KUKA KRL program: PPR_fullpath_2mm_split3.src

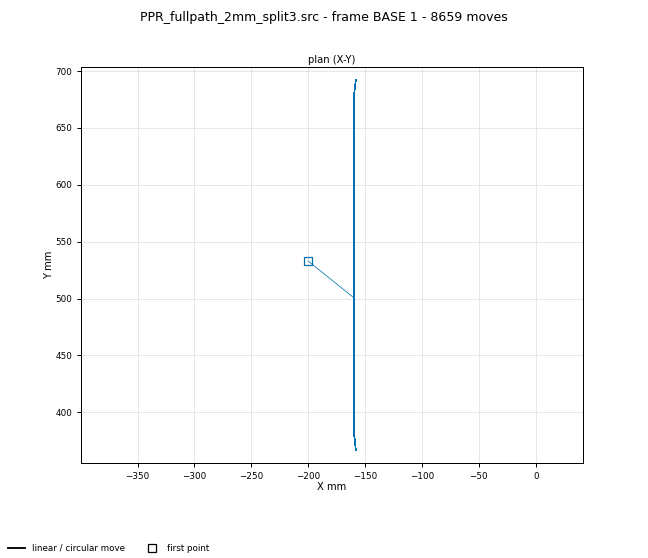
[picture p0: tool path of PPR_fullpath_2mm_split3.src in frame BASE 1, 8659 of 8660 moves have a stored position in this frame; points joined in program order, loops and branches not executed]
&ACCESS RVEO
&REL 11
&PARAM TEMPLATE = C:\KRC\Roboter\Template\vorgabe
&PARAM EDITMASK = *
DEF variable_helical2( )
;FOLD INI
  ;FOLD BASISTECH INI
    GLOBAL INTERRUPT DECL 3 WHEN $STOPMESS==TRUE DO IR_STOPM ( )
    INTERRUPT ON 3
    BAS (#INITMOV,0 )
  ;ENDFOLD (BASISTECH INI)
 ;FOLD USER INI


    ;Make your modifications here
  ;ENDFOLD (USER INI)
;ENDFOLD (INI)
ACTION(#AXIS_RESET,34,1000,#NOERROR,ERROR_CODE)
;FOLD PTP HOME  Vel= 100 % DEFAULT;%{PE}%MKUKATPBASIS,%CMOVE,%VPTP,%P 1:PTP, 2:HOME, 3:, 5:100, 7:DEFAULT
$BWDSTART = FALSE
PDAT_ACT=PDEFAULT
FDAT_ACT=FHOME
BAS (#PTP_PARAMS,100 )
$H_POS=XHOME
PTP  XHOME
;ENDFOLD
BAS(#TOOL,1)
BAS(#BASE,1)
$VEL_AXIS[1]=100
$VEL_AXIS[2]=100
$VEL_AXIS[3]=100
$VEL_AXIS[4]=100
$VEL_AXIS[5]=100
$VEL_AXIS[6]=100
$VEL_EXTAX[1]=100
$VEL_EXTAX[2]=100

$ACC_AXIS[1]=100
$ACC_AXIS[2]=100
$ACC_AXIS[3]=100
$ACC_AXIS[4]=100
$ACC_AXIS[5]=100
$ACC_AXIS[6]=100
$ACC_EXTAX[1]=100
$ACC_EXTAX[2]=100

SLIN {X  -200.000, Y  +533.000, Z    +0.000, A    +0.000, E1    +0.000, E3    +0.000, E4    +0.000}

SLIN {X  -160.000, Y  +500.804, Z    +0.000, E1   +21.423, E3  -369.741}
HALT
SPLINE
SPL {X  -160.000, Y  +497.229, Z    +0.000, E1   +21.403, E3  -350.308}
SPL {X  -160.000, Y  +493.901, Z    +0.000, E1   +21.409, E3  -332.289}
SPL {X  -160.000, Y  +490.791, Z    +0.000, E1   +21.400, E3  -315.416}
SPL {X  -160.000, Y  +487.647, Z    +0.000, E1   +21.401, E3  -298.370}
SPL {X  -160.000, Y  +484.273, Z    +0.000, E1   +21.408, E3  -280.090}
SPL {X  -160.000, Y  +481.093, Z    +0.000, E1   +21.389, E3  -262.781}
SPL {X  -160.000, Y  +478.021, Z    +0.000, E1   +21.401, E3  -246.174}
SPL {X  -160.000, Y  +474.639, Z    +0.000, E1   +21.410, E3  -227.883}
SPL {X  -160.000, Y  +471.343, Z    +0.000, E1   +21.399, E3  -209.981}
SPL {X  -160.000, Y  +468.133, Z    +0.000, E1   +21.402, E3  -192.589}
SPL {X  -160.000, Y  +464.638, Z    +0.000, E1   +21.421, E3  -173.740}
SPL {X  -160.000, Y  +461.045, Z    +0.000, E1   +21.424, E3  -154.326}
SPL {X  -160.000, Y  +457.606, Z    +0.000, E1   +21.413, E3  -135.616}
SPL {X  -160.000, Y  +454.417, Z    +0.000, E1   +21.401, E3  -118.308}
SPL {X  -160.000, Y  +451.425, Z    +0.000, E1   +21.404, E3  -102.086}
SPL {X  -160.000, Y  +448.039, Z    +0.000, E1   +21.417, E3   -83.793}
SPL {X  -160.000, Y  +444.787, Z    +0.000, E1   +21.414, E3   -66.238}
SPL {X  -160.000, Y  +441.637, Z    +0.000, E1   +21.431, E3   -49.260}
SPL {X  -160.000, Y  +438.199, Z    +0.000, E1   +21.432, E3   -30.656}
SPL {X  -160.000, Y  +434.875, Z    +0.000, E1   +21.424, E3   -12.616}
SPL {X  -160.000, Y  +431.689, Z    +0.000, E1   +21.423, E3    +4.632}
SPL {X  -160.000, Y  +428.451, Z    +0.000, E1   +21.430, E3   +22.112}
SPL {X  -160.000, Y  +425.120, Z    +0.000, E1   +21.430, E3   +40.176}
SPL {X  -160.000, Y  +421.671, Z    +0.000, E1   +21.430, E3   +58.860}
SPL {X  -160.000, Y  +418.225, Z    +0.000, E1   +21.425, E3   +77.542}
SPL {X  -160.000, Y  +414.956, Z    +0.000, E1   +21.424, E3   +95.222}
SPL {X  -160.000, Y  +411.834, Z    +0.000, E1   +21.420, E3  +112.140}
SPL {X  -160.000, Y  +408.570, Z    +0.000, E1   +21.432, E3  +129.749}
SPL {X  -160.000, Y  +405.237, Z    +0.000, E1   +21.432, E3  +147.778}
SPL {X  -160.000, Y  +402.004, Z    +0.000, E1   +21.424, E3  +165.353}
SPL {X  -160.000, Y  +398.626, Z    +0.000, E1   +21.425, E3  +183.659}
SPL {X  -160.000, Y  +395.405, Z    +0.000, E1   +21.422, E3  +201.077}
SPL {X  -160.000, Y  +392.641, Z    +0.000, E1   +21.407, E3  +216.075}
SPL {X  -159.989, Y  +390.129, Z    +0.000, E1   +21.406, E3  +229.716}
SPL {X  -159.932, Y  +387.337, Z    +0.000, E1   +21.403, E3  +244.912}
SPL {X  -159.823, Y  +384.478, Z    +0.000, E1   +21.379, E3  +260.575}
SPL {X  -159.660, Y  +381.581, Z    +0.000, E1   +21.363, E3  +276.463}
SPL {X  -159.452, Y  +378.773, Z    +0.000, E1   +21.330, E3  +291.910}
SPL {X  -159.222, Y  +376.244, Z    +0.000, E1   +21.297, E3  +305.872}
SPL {X  -158.814, Y  +372.556, Z    +0.000, E1   +21.316, E3  +326.139}
SPL {X  -158.301, Y  +368.743, Z    +0.000, E1   +21.199, E3  +347.461}
SPL {X  -157.981, Y  +366.660, Z    +0.000, E1   +19.986, E3  +370.429}
ENDSPLINE

SPLINE
SPL {X  -158.491, Y  +370.077, Z    +0.000, E1   +15.910, E3  +395.442}
SPL {X  -159.771, Y  +383.450, Z    +0.000, E1    +6.314, E3  +418.597}
SPL {X  -160.000, Y  +392.463, Z    +0.000, E1    +0.112, E3  +425.104}
SPL {X  -160.000, Y  +399.874, Z    +0.000, E1    -5.508, E3  +429.606}
SPL {X  -160.000, Y  +411.622, Z    +0.000, E1   -13.815, E3  +441.726}
SPL {X  -160.000, Y  +419.836, Z    +0.000, E1   -18.198, E3  +456.900}
SPL {X  -160.000, Y  +430.523, Z    +0.000, E1   -21.710, E3  +487.100}
SPL {X  -160.000, Y  +433.426, Z    +0.000, E1   -21.735, E3  +502.515}
SPL {X  -160.000, Y  +436.131, Z    +0.000, E1   -21.710, E3  +516.989}
SPL {X  -160.000, Y  +439.046, Z    +0.000, E1   -21.732, E3  +532.483}
SPL {X  -160.000, Y  +442.009, Z    +0.000, E1   -21.719, E3  +548.305}
SPL {X  -160.000, Y  +444.891, Z    +0.000, E1   -21.724, E3  +563.661}
SPL {X  -160.000, Y  +449.017, Z    +0.000, E1   -21.792, E3  +585.452}
SPL {X  -160.000, Y  +452.864, Z    +0.000, E1   -21.730, E3  +606.070}
SPL {X  -160.000, Y  +455.470, Z    +0.000, E1   -21.722, E3  +619.959}
SPL {X  -160.000, Y  +458.295, Z    +0.000, E1   -21.738, E3  +634.980}
SPL {X  -160.000, Y  +461.133, Z    +0.000, E1   -21.720, E3  +650.162}
SPL {X  -160.000, Y  +464.458, Z    +0.000, E1   -21.770, E3  +667.681}
SPL {X  -160.000, Y  +468.250, Z    +0.000, E1   -21.764, E3  +687.834}
SPL {X  -160.000, Y  +472.226, Z    +0.000, E1   -21.782, E3  +708.993}
SPL {X  -160.000, Y  +476.333, Z    +0.000, E1   -21.767, E3  +730.907}
SPL {X  -160.000, Y  +480.244, Z    +0.000, E1   -21.765, E3  +751.772}
SPL {X  -160.000, Y  +484.301, Z    +0.000, E1   -21.775, E3  +773.300}
SPL {X  -160.000, Y  +488.201, Z    +0.000, E1   -21.768, E3  +794.060}
SPL {X  -160.000, Y  +492.394, Z    +0.000, E1   -21.802, E3  +816.234}
SPL {X  -160.000, Y  +496.781, Z    +0.000, E1   -21.798, E3  +839.546}
SPL {X  -160.000, Y  +501.083, Z    +0.000, E1   -21.796, E3  +862.476}
SPL {X  -160.000, Y  +504.917, Z    +0.000, E1   -21.764, E3  +882.980}
SPL {X  -160.000, Y  +508.886, Z    +0.000, E1   -21.791, E3  +904.066}
SPL {X  -160.000, Y  +513.057, Z    +0.000, E1   -21.767, E3  +926.374}
SPL {X  -160.000, Y  +517.221, Z    +0.000, E1   -21.778, E3  +948.527}
SPL {X  -160.000, Y  +521.677, Z    +0.000, E1   -21.781, E3  +972.288}
SPL {X  -160.000, Y  +525.729, Z    +0.000, E1   -21.753, E3  +993.927}
SPL {X  -160.000, Y  +529.456, Z    +0.000, E1   -21.766, E3 +1013.706}
SPL {X  -160.000, Y  +533.608, Z    +0.000, E1   -21.776, E3 +1035.837}
SPL {X  -160.000, Y  +538.227, Z    +0.000, E1   -21.794, E3 +1060.369}
SPL {X  -160.000, Y  +542.483, Z    +0.000, E1   -21.764, E3 +1083.095}
SPL {X  -160.000, Y  +546.194, Z    +0.000, E1   -21.754, E3 +1102.911}
SPL {X  -160.000, Y  +550.131, Z    +0.000, E1   -21.771, E3 +1123.847}
SPL {X  -160.000, Y  +554.462, Z    +0.000, E1   -21.777, E3 +1146.901}
SPL {X  -160.000, Y  +558.542, Z    +0.000, E1   -21.758, E3 +1168.673}
SPL {X  -160.000, Y  +562.615, Z    +0.000, E1   -21.776, E3 +1190.329}
SPL {X  -160.000, Y  +566.764, Z    +0.000, E1   -21.764, E3 +1212.454}
SPL {X  -160.000, Y  +570.657, Z    +0.000, E1   -21.758, E3 +1233.201}
SPL {X  -160.000, Y  +574.688, Z    +0.000, E1   -21.771, E3 +1254.644}
SPL {X  -160.000, Y  +578.864, Z    +0.000, E1   -21.770, E3 +1276.895}
SPL {X  -160.000, Y  +582.807, Z    +0.000, E1   -21.754, E3 +1297.949}
SPL {X  -160.000, Y  +586.993, Z    +0.000, E1   -21.779, E3 +1320.185}
SPL {X  -160.000, Y  +591.368, Z    +0.000, E1   -21.775, E3 +1343.472}
SPL {X  -160.000, Y  +595.703, Z    +0.000, E1   -21.775, E3 +1366.581}
SPL {X  -160.000, Y  +599.558, Z    +0.000, E1   -21.748, E3 +1387.159}
SPL {X  -160.000, Y  +603.126, Z    +0.000, E1   -21.757, E3 +1406.138}
SPL {X  -160.000, Y  +607.107, Z    +0.000, E1   -21.766, E3 +1427.364}
SPL {X  -160.000, Y  +611.246, Z    +0.000, E1   -21.760, E3 +1449.437}
SPL {X  -160.000, Y  +615.151, Z    +0.000, E1   -21.752, E3 +1470.250}
SPL {X  -160.000, Y  +618.728, Z    +0.000, E1   -21.747, E3 +1489.312}
SPL {X  -160.000, Y  +622.318, Z    +0.000, E1   -21.753, E3 +1508.427}
SPL {X  -160.000, Y  +625.877, Z    +0.000, E1   -21.745, E3 +1527.405}
SPL {X  -160.000, Y  +629.892, Z    +0.000, E1   -21.777, E3 +1548.729}
SPL {X  -160.000, Y  +634.024, Z    +0.000, E1   -21.756, E3 +1570.779}
SPL {X  -160.000, Y  +637.661, Z    +0.000, E1   -21.748, E3 +1590.170}
SPL {X  -160.000, Y  +641.244, Z    +0.000, E1   -21.752, E3 +1609.241}
SPL {X  -160.000, Y  +645.120, Z    +0.000, E1   -21.762, E3 +1629.873}
SPL {X  -160.000, Y  +649.214, Z    +0.000, E1   -21.766, E3 +1651.661}
SPL {X  -160.000, Y  +653.188, Z    +0.000, E1   -21.771, E3 +1672.724}
SPL {X  -160.000, Y  +656.905, Z    +0.000, E1   -21.769, E3 +1692.499}
SPL {X  -160.000, Y  +660.685, Z    +0.000, E1   -21.769, E3 +1712.667}
SPL {X  -160.000, Y  +664.985, Z    +0.000, E1   -21.790, E3 +1735.520}
SPL {X  -159.993, Y  +669.170, Z    +0.000, E1   -21.763, E3 +1757.878}
SPL {X  -159.916, Y  +672.869, Z    +0.000, E1   -21.755, E3 +1777.623}
SPL {X  -159.752, Y  +676.610, Z    +0.000, E1   -21.740, E3 +1797.698}
SPL {X  -159.478, Y  +680.618, Z    +0.000, E1   -21.719, E3 +1819.297}
SPL {X  -159.108, Y  +684.576, Z    +0.000, E1   -21.664, E3 +1840.767}
SPL {X  -158.638, Y  +688.530, Z    +0.000, E1   -21.617, E3 +1862.288}
SPL {X  -158.097, Y  +692.303, Z    +0.000, E1   -21.529, E3 +1883.006}
ENDSPLINE

SPLINE
SPL {X  -158.264, Y  +691.203, Z    +0.000, E1   -17.264, E3 +1919.751}
SPL {X  -159.000, Y  +685.560, Z    +0.000, E1   -12.398, E3 +1940.927}
SPL {X  -159.924, Y  +672.625, Z    +0.000, E1    -3.689, E3 +1955.944}
SPL {X  -160.000, Y  +663.203, Z    +0.000, E1    +3.155, E3 +1962.598}
SPL {X  -160.000, Y  +652.103, Z    +0.000, E1   +11.247, E3 +1974.268}
SPL {X  -160.000, Y  +641.822, Z    +0.000, E1   +17.059, E3 +1993.642}
SPL {X  -160.000, Y  +631.293, Z    +0.000, E1   +20.354, E3 +2027.522}
SPL {X  -160.000, Y  +627.542, Z    +0.000, E1   +20.380, E3 +2048.929}
SPL {X  -160.000, Y  +623.532, Z    +0.000, E1   +20.378, E3 +2071.894}
SPL {X  -160.000, Y  +619.329, Z    +0.000, E1   +20.391, E3 +2095.932}
SPL {X  -160.000, Y  +614.967, Z    +0.000, E1   +20.392, E3 +2120.912}
SPL {X  -160.000, Y  +611.206, Z    +0.000, E1   +20.351, E3 +2142.583}
SPL {X  -160.000, Y  +607.824, Z    +0.000, E1   +20.354, E3 +2162.004}
SPL {X  -160.000, Y  +603.899, Z    +0.000, E1   +20.373, E3 +2184.454}
SPL {X  -160.000, Y  +599.617, Z    +0.000, E1   +20.384, E3 +2208.948}
SPL {X  -160.000, Y  +595.532, Z    +0.000, E1   +20.373, E3 +2232.308}
SPL {X  -160.000, Y  +591.705, Z    +0.000, E1   +20.373, E3 +2254.233}
SPL {X  -160.000, Y  +588.037, Z    +0.000, E1   +20.359, E3 +2275.320}
SPL {X  -160.000, Y  +584.320, Z    +0.000, E1   +20.364, E3 +2296.622}
SPL {X  -160.000, Y  +580.616, Z    +0.000, E1   +20.357, E3 +2317.849}
SPL {X  -160.000, Y  +577.083, Z    +0.000, E1   +20.358, E3 +2338.097}
SPL {X  -160.000, Y  +573.158, Z    +0.000, E1   +20.377, E3 +2360.549}
SPL {X  -160.000, Y  +568.802, Z    +0.000, E1   +20.385, E3 +2385.501}
SPL {X  -160.000, Y  +564.937, Z    +0.000, E1   +20.350, E3 +2407.722}
SPL {X  -160.000, Y  +561.213, Z    +0.000, E1   +20.372, E3 +2429.008}
SPL {X  -160.000, Y  +557.320, Z    +0.000, E1   +20.363, E3 +2451.335}
SPL {X  -160.000, Y  +553.712, Z    +0.000, E1   +20.355, E3 +2472.034}
SPL {X  -160.000, Y  +550.040, Z    +0.000, E1   +20.360, E3 +2493.072}
SPL {X  -160.000, Y  +546.180, Z    +0.000, E1   +20.370, E3 +2515.128}
SPL {X  -160.000, Y  +542.032, Z    +0.000, E1   +20.384, E3 +2538.867}
SPL {X  -160.000, Y  +537.870, Z    +0.000, E1   +20.372, E3 +2562.743}
SPL {X  -160.000, Y  +534.086, Z    +0.000, E1   +20.356, E3 +2584.497}
SPL {X  -160.000, Y  +530.164, Z    +0.000, E1   +20.382, E3 +2606.846}
SPL {X  -160.000, Y  +527.505, Z    +0.000, E1   +20.318, E3 +2622.220}
SPL {X  -160.000, Y  +511.620, Z    +0.000, E1   +28.365, E3 +2632.683}
SPL {X  -160.000, Y  +507.906, Z    +0.000, E1   +28.152, E3 +2649.078}
SPL {X  -160.000, Y  +506.085, Z    +0.000, E1   +26.146, E3 +2671.538}
SPL {X  -160.000, Y  +504.342, Z    +0.000, E1   +24.109, E3 +2695.053}
SPL {X  -160.000, Y  +503.002, Z    +0.000, E1   +22.325, E3 +2716.058}
SPL {X  -160.000, Y  +500.783, Z    +0.000, E1   +21.421, E3 +2735.647}
SPL {X  -160.000, Y  +497.229, Z    +0.000, E1   +21.403, E3 +2754.956}
SPL {X  -160.000, Y  +493.901, Z    +0.000, E1   +21.409, E3 +2772.975}
SPL {X  -160.000, Y  +490.791, Z    +0.000, E1   +21.400, E3 +2789.848}
SPL {X  -160.000, Y  +487.647, Z    +0.000, E1   +21.401, E3 +2806.894}
SPL {X  -160.000, Y  +484.273, Z    +0.000, E1   +21.408, E3 +2825.174}
SPL {X  -160.000, Y  +481.093, Z    +0.000, E1   +21.389, E3 +2842.483}
SPL {X  -160.000, Y  +478.021, Z    +0.000, E1   +21.401, E3 +2859.089}
SPL {X  -160.000, Y  +474.639, Z    +0.000, E1   +21.410, E3 +2877.381}
SPL {X  -160.000, Y  +471.343, Z    +0.000, E1   +21.399, E3 +2895.283}
SPL {X  -160.000, Y  +468.133, Z    +0.000, E1   +21.402, E3 +2912.674}
SPL {X  -160.000, Y  +464.638, Z    +0.000, E1   +21.421, E3 +2931.523}
SPL {X  -160.000, Y  +461.045, Z    +0.000, E1   +21.424, E3 +2950.937}
SPL {X  -160.000, Y  +457.606, Z    +0.000, E1   +21.413, E3 +2969.647}
SPL {X  -160.000, Y  +454.417, Z    +0.000, E1   +21.401, E3 +2986.956}
SPL {X  -160.000, Y  +451.425, Z    +0.000, E1   +21.404, E3 +3003.177}
SPL {X  -160.000, Y  +448.039, Z    +0.000, E1   +21.417, E3 +3021.470}
SPL {X  -160.000, Y  +444.787, Z    +0.000, E1   +21.414, E3 +3039.025}
SPL {X  -160.000, Y  +441.637, Z    +0.000, E1   +21.431, E3 +3056.004}
SPL {X  -160.000, Y  +438.199, Z    +0.000, E1   +21.432, E3 +3074.607}
SPL {X  -160.000, Y  +434.875, Z    +0.000, E1   +21.424, E3 +3092.647}
SPL {X  -160.000, Y  +431.689, Z    +0.000, E1   +21.423, E3 +3109.896}
SPL {X  -160.000, Y  +428.451, Z    +0.000, E1   +21.430, E3 +3127.375}
SPL {X  -160.000, Y  +425.120, Z    +0.000, E1   +21.430, E3 +3145.440}
SPL {X  -160.000, Y  +421.671, Z    +0.000, E1   +21.430, E3 +3164.123}
SPL {X  -160.000, Y  +418.225, Z    +0.000, E1   +21.425, E3 +3182.805}
SPL {X  -160.000, Y  +414.956, Z    +0.000, E1   +21.424, E3 +3200.486}
SPL {X  -160.000, Y  +411.834, Z    +0.000, E1   +21.420, E3 +3217.404}
SPL {X  -160.000, Y  +408.570, Z    +0.000, E1   +21.432, E3 +3235.013}
SPL {X  -160.000, Y  +405.237, Z    +0.000, E1   +21.432, E3 +3253.041}
SPL {X  -160.000, Y  +402.004, Z    +0.000, E1   +21.424, E3 +3270.617}
SPL {X  -160.000, Y  +398.626, Z    +0.000, E1   +21.425, E3 +3288.923}
SPL {X  -160.000, Y  +395.405, Z    +0.000, E1   +21.422, E3 +3306.340}
SPL {X  -160.000, Y  +392.641, Z    +0.000, E1   +21.407, E3 +3321.339}
SPL {X  -159.989, Y  +390.129, Z    +0.000, E1   +21.406, E3 +3334.980}
SPL {X  -159.932, Y  +387.337, Z    +0.000, E1   +21.403, E3 +3350.175}
SPL {X  -159.823, Y  +384.478, Z    +0.000, E1   +21.379, E3 +3365.838}
SPL {X  -159.660, Y  +381.581, Z    +0.000, E1   +21.363, E3 +3381.727}
SPL {X  -159.452, Y  +378.773, Z    +0.000, E1   +21.330, E3 +3397.173}
SPL {X  -159.222, Y  +376.244, Z    +0.000, E1   +21.297, E3 +3411.136}
SPL {X  -158.814, Y  +372.556, Z    +0.000, E1   +21.316, E3 +3431.403}
SPL {X  -158.301, Y  +368.743, Z    +0.000, E1   +21.199, E3 +3452.725}
SPL {X  -157.981, Y  +366.660, Z    +0.000, E1   +19.986, E3 +3475.692}
ENDSPLINE

SPLINE
SPL {X  -158.491, Y  +370.077, Z    +0.000, E1   +15.910, E3 +3500.705}
SPL {X  -159.771, Y  +383.450, Z    +0.000, E1    +6.314, E3 +3523.861}
SPL {X  -160.000, Y  +392.463, Z    +0.000, E1    +0.112, E3 +3530.367}
SPL {X  -160.000, Y  +399.874, Z    +0.000, E1    -5.508, E3 +3534.870}
SPL {X  -160.000, Y  +411.622, Z    +0.000, E1   -13.815, E3 +3546.990}
SPL {X  -160.000, Y  +419.836, Z    +0.000, E1   -18.198, E3 +3562.163}
SPL {X  -160.000, Y  +430.523, Z    +0.000, E1   -21.710, E3 +3592.364}
SPL {X  -160.000, Y  +433.426, Z    +0.000, E1   -21.735, E3 +3607.778}
SPL {X  -160.000, Y  +436.131, Z    +0.000, E1   -21.710, E3 +3622.253}
SPL {X  -160.000, Y  +439.046, Z    +0.000, E1   -21.732, E3 +3637.746}
SPL {X  -160.000, Y  +442.009, Z    +0.000, E1   -21.719, E3 +3653.568}
SPL {X  -160.000, Y  +444.891, Z    +0.000, E1   -21.724, E3 +3668.924}
SPL {X  -160.000, Y  +449.017, Z    +0.000, E1   -21.792, E3 +3690.716}
SPL {X  -160.000, Y  +452.864, Z    +0.000, E1   -21.730, E3 +3711.333}
SPL {X  -160.000, Y  +455.470, Z    +0.000, E1   -21.722, E3 +3725.222}
SPL {X  -160.000, Y  +458.295, Z    +0.000, E1   -21.738, E3 +3740.243}
SPL {X  -160.000, Y  +461.133, Z    +0.000, E1   -21.720, E3 +3755.426}
SPL {X  -160.000, Y  +464.458, Z    +0.000, E1   -21.770, E3 +3772.945}
SPL {X  -160.000, Y  +468.250, Z    +0.000, E1   -21.764, E3 +3793.098}
SPL {X  -160.000, Y  +472.226, Z    +0.000, E1   -21.782, E3 +3814.256}
SPL {X  -160.000, Y  +476.333, Z    +0.000, E1   -21.767, E3 +3836.171}
SPL {X  -160.000, Y  +480.244, Z    +0.000, E1   -21.765, E3 +3857.035}
SPL {X  -160.000, Y  +484.301, Z    +0.000, E1   -21.775, E3 +3878.564}
SPL {X  -160.000, Y  +488.201, Z    +0.000, E1   -21.768, E3 +3899.324}
SPL {X  -160.000, Y  +492.394, Z    +0.000, E1   -21.802, E3 +3921.498}
SPL {X  -160.000, Y  +496.781, Z    +0.000, E1   -21.798, E3 +3944.809}
SPL {X  -160.000, Y  +501.083, Z    +0.000, E1   -21.796, E3 +3967.739}
SPL {X  -160.000, Y  +504.917, Z    +0.000, E1   -21.764, E3 +3988.244}
SPL {X  -160.000, Y  +508.886, Z    +0.000, E1   -21.791, E3 +4009.330}
SPL {X  -160.000, Y  +513.057, Z    +0.000, E1   -21.767, E3 +4031.637}
SPL {X  -160.000, Y  +517.221, Z    +0.000, E1   -21.778, E3 +4053.790}
SPL {X  -160.000, Y  +521.677, Z    +0.000, E1   -21.781, E3 +4077.551}
SPL {X  -160.000, Y  +525.729, Z    +0.000, E1   -21.753, E3 +4099.191}
SPL {X  -160.000, Y  +529.456, Z    +0.000, E1   -21.766, E3 +4118.970}
SPL {X  -160.000, Y  +533.608, Z    +0.000, E1   -21.776, E3 +4141.100}
SPL {X  -160.000, Y  +538.227, Z    +0.000, E1   -21.794, E3 +4165.633}
SPL {X  -160.000, Y  +542.483, Z    +0.000, E1   -21.764, E3 +4188.358}
SPL {X  -160.000, Y  +546.194, Z    +0.000, E1   -21.754, E3 +4208.174}
SPL {X  -160.000, Y  +550.131, Z    +0.000, E1   -21.771, E3 +4229.110}
SPL {X  -160.000, Y  +554.462, Z    +0.000, E1   -21.777, E3 +4252.164}
SPL {X  -160.000, Y  +558.542, Z    +0.000, E1   -21.758, E3 +4273.937}
SPL {X  -160.000, Y  +562.615, Z    +0.000, E1   -21.776, E3 +4295.593}
SPL {X  -160.000, Y  +566.764, Z    +0.000, E1   -21.764, E3 +4317.718}
SPL {X  -160.000, Y  +570.657, Z    +0.000, E1   -21.758, E3 +4338.465}
SPL {X  -160.000, Y  +574.688, Z    +0.000, E1   -21.771, E3 +4359.908}
SPL {X  -160.000, Y  +578.864, Z    +0.000, E1   -21.770, E3 +4382.159}
SPL {X  -160.000, Y  +582.807, Z    +0.000, E1   -21.754, E3 +4403.213}
SPL {X  -160.000, Y  +586.993, Z    +0.000, E1   -21.779, E3 +4425.448}
SPL {X  -160.000, Y  +591.368, Z    +0.000, E1   -21.775, E3 +4448.735}
SPL {X  -160.000, Y  +595.703, Z    +0.000, E1   -21.775, E3 +4471.845}
SPL {X  -160.000, Y  +599.558, Z    +0.000, E1   -21.748, E3 +4492.422}
SPL {X  -160.000, Y  +603.126, Z    +0.000, E1   -21.757, E3 +4511.402}
SPL {X  -160.000, Y  +607.107, Z    +0.000, E1   -21.766, E3 +4532.627}
SPL {X  -160.000, Y  +611.246, Z    +0.000, E1   -21.760, E3 +4554.700}
SPL {X  -160.000, Y  +615.151, Z    +0.000, E1   -21.752, E3 +4575.514}
SPL {X  -160.000, Y  +618.728, Z    +0.000, E1   -21.747, E3 +4594.576}
SPL {X  -160.000, Y  +622.318, Z    +0.000, E1   -21.753, E3 +4613.690}
SPL {X  -160.000, Y  +625.877, Z    +0.000, E1   -21.745, E3 +4632.669}
SPL {X  -160.000, Y  +629.892, Z    +0.000, E1   -21.777, E3 +4653.992}
SPL {X  -160.000, Y  +634.024, Z    +0.000, E1   -21.756, E3 +4676.043}
SPL {X  -160.000, Y  +637.661, Z    +0.000, E1   -21.748, E3 +4695.433}
SPL {X  -160.000, Y  +641.244, Z    +0.000, E1   -21.752, E3 +4714.504}
SPL {X  -160.000, Y  +645.120, Z    +0.000, E1   -21.762, E3 +4735.137}
SPL {X  -160.000, Y  +649.214, Z    +0.000, E1   -21.766, E3 +4756.925}
SPL {X  -160.000, Y  +653.188, Z    +0.000, E1   -21.771, E3 +4777.987}
SPL {X  -160.000, Y  +656.905, Z    +0.000, E1   -21.769, E3 +4797.763}
SPL {X  -160.000, Y  +660.685, Z    +0.000, E1   -21.769, E3 +4817.931}
SPL {X  -160.000, Y  +664.985, Z    +0.000, E1   -21.790, E3 +4840.783}
SPL {X  -159.993, Y  +669.170, Z    +0.000, E1   -21.763, E3 +4863.142}
SPL {X  -159.916, Y  +672.869, Z    +0.000, E1   -21.755, E3 +4882.887}
SPL {X  -159.752, Y  +676.610, Z    +0.000, E1   -21.740, E3 +4902.962}
SPL {X  -159.478, Y  +680.618, Z    +0.000, E1   -21.719, E3 +4924.561}
SPL {X  -159.108, Y  +684.576, Z    +0.000, E1   -21.664, E3 +4946.030}
SPL {X  -158.638, Y  +688.530, Z    +0.000, E1   -21.617, E3 +4967.552}
SPL {X  -158.097, Y  +692.303, Z    +0.000, E1   -21.529, E3 +4988.269}
ENDSPLINE

SPLINE
SPL {X  -158.264, Y  +691.203, Z    +0.000, E1   -17.264, E3 +5025.015}
SPL {X  -159.000, Y  +685.560, Z    +0.000, E1   -12.398, E3 +5046.190}
SPL {X  -159.924, Y  +672.625, Z    +0.000, E1    -3.689, E3 +5061.207}
SPL {X  -160.000, Y  +663.203, Z    +0.000, E1    +3.155, E3 +5067.862}
SPL {X  -160.000, Y  +652.103, Z    +0.000, E1   +11.247, E3 +5079.532}
SPL {X  -160.000, Y  +641.822, Z    +0.000, E1   +17.059, E3 +5098.906}
SPL {X  -160.000, Y  +631.293, Z    +0.000, E1   +20.354, E3 +5132.785}
SPL {X  -160.000, Y  +627.542, Z    +0.000, E1   +20.380, E3 +5154.192}
SPL {X  -160.000, Y  +623.532, Z    +0.000, E1   +20.378, E3 +5177.158}
SPL {X  -160.000, Y  +619.329, Z    +0.000, E1   +20.391, E3 +5201.195}
SPL {X  -160.000, Y  +614.967, Z    +0.000, E1   +20.392, E3 +5226.175}
SPL {X  -160.000, Y  +611.206, Z    +0.000, E1   +20.351, E3 +5247.847}
SPL {X  -160.000, Y  +607.824, Z    +0.000, E1   +20.354, E3 +5267.268}
SPL {X  -160.000, Y  +603.899, Z    +0.000, E1   +20.373, E3 +5289.718}
SPL {X  -160.000, Y  +599.617, Z    +0.000, E1   +20.384, E3 +5314.212}
SPL {X  -160.000, Y  +595.532, Z    +0.000, E1   +20.373, E3 +5337.572}
SPL {X  -160.000, Y  +591.705, Z    +0.000, E1   +20.373, E3 +5359.497}
SPL {X  -160.000, Y  +588.037, Z    +0.000, E1   +20.359, E3 +5380.584}
SPL {X  -160.000, Y  +584.320, Z    +0.000, E1   +20.364, E3 +5401.885}
SPL {X  -160.000, Y  +580.616, Z    +0.000, E1   +20.357, E3 +5423.112}
SPL {X  -160.000, Y  +577.083, Z    +0.000, E1   +20.358, E3 +5443.361}
SPL {X  -160.000, Y  +573.158, Z    +0.000, E1   +20.377, E3 +5465.813}
SPL {X  -160.000, Y  +568.802, Z    +0.000, E1   +20.385, E3 +5490.765}
SPL {X  -160.000, Y  +564.937, Z    +0.000, E1   +20.350, E3 +5512.985}
SPL {X  -160.000, Y  +561.213, Z    +0.000, E1   +20.372, E3 +5534.272}
SPL {X  -160.000, Y  +557.320, Z    +0.000, E1   +20.363, E3 +5556.598}
SPL {X  -160.000, Y  +553.712, Z    +0.000, E1   +20.355, E3 +5577.298}
SPL {X  -160.000, Y  +550.040, Z    +0.000, E1   +20.360, E3 +5598.336}
SPL {X  -160.000, Y  +546.180, Z    +0.000, E1   +20.370, E3 +5620.392}
SPL {X  -160.000, Y  +542.032, Z    +0.000, E1   +20.384, E3 +5644.131}
SPL {X  -160.000, Y  +537.870, Z    +0.000, E1   +20.372, E3 +5668.006}
SPL {X  -160.000, Y  +534.086, Z    +0.000, E1   +20.356, E3 +5689.760}
SPL {X  -160.000, Y  +530.164, Z    +0.000, E1   +20.382, E3 +5712.110}
SPL {X  -160.000, Y  +527.505, Z    +0.000, E1   +20.318, E3 +5727.484}
SPL {X  -160.000, Y  +511.620, Z    +0.000, E1   +28.365, E3 +5737.947}
SPL {X  -160.000, Y  +507.906, Z    +0.000, E1   +28.152, E3 +5754.342}
SPL {X  -160.000, Y  +506.085, Z    +0.000, E1   +26.146, E3 +5776.801}
SPL {X  -160.000, Y  +504.342, Z    +0.000, E1   +24.109, E3 +5800.316}
SPL {X  -160.000, Y  +503.002, Z    +0.000, E1   +22.325, E3 +5821.322}
SPL {X  -160.000, Y  +500.783, Z    +0.000, E1   +21.421, E3 +5840.911}
SPL {X  -160.000, Y  +497.229, Z    +0.000, E1   +21.403, E3 +5860.219}
SPL {X  -160.000, Y  +493.901, Z    +0.000, E1   +21.409, E3 +5878.238}
SPL {X  -160.000, Y  +490.791, Z    +0.000, E1   +21.400, E3 +5895.111}
SPL {X  -160.000, Y  +487.647, Z    +0.000, E1   +21.401, E3 +5912.157}
SPL {X  -160.000, Y  +484.273, Z    +0.000, E1   +21.408, E3 +5930.437}
SPL {X  -160.000, Y  +481.093, Z    +0.000, E1   +21.389, E3 +5947.746}
SPL {X  -160.000, Y  +478.021, Z    +0.000, E1   +21.401, E3 +5964.353}
SPL {X  -160.000, Y  +474.639, Z    +0.000, E1   +21.410, E3 +5982.644}
SPL {X  -160.000, Y  +471.343, Z    +0.000, E1   +21.399, E3 +6000.546}
SPL {X  -160.000, Y  +468.133, Z    +0.000, E1   +21.402, E3 +6017.938}
SPL {X  -160.000, Y  +464.638, Z    +0.000, E1   +21.421, E3 +6036.787}
SPL {X  -160.000, Y  +461.045, Z    +0.000, E1   +21.424, E3 +6056.201}
SPL {X  -160.000, Y  +457.606, Z    +0.000, E1   +21.413, E3 +6074.911}
SPL {X  -160.000, Y  +454.417, Z    +0.000, E1   +21.401, E3 +6092.219}
SPL {X  -160.000, Y  +451.425, Z    +0.000, E1   +21.404, E3 +6108.441}
SPL {X  -160.000, Y  +448.039, Z    +0.000, E1   +21.417, E3 +6126.734}
SPL {X  -160.000, Y  +444.787, Z    +0.000, E1   +21.414, E3 +6144.289}
SPL {X  -160.000, Y  +441.637, Z    +0.000, E1   +21.431, E3 +6161.267}
SPL {X  -160.000, Y  +438.199, Z    +0.000, E1   +21.432, E3 +6179.871}
SPL {X  -160.000, Y  +434.875, Z    +0.000, E1   +21.424, E3 +6197.911}
SPL {X  -160.000, Y  +431.689, Z    +0.000, E1   +21.423, E3 +6215.159}
SPL {X  -160.000, Y  +428.451, Z    +0.000, E1   +21.430, E3 +6232.639}
SPL {X  -160.000, Y  +425.120, Z    +0.000, E1   +21.430, E3 +6250.703}
SPL {X  -160.000, Y  +421.671, Z    +0.000, E1   +21.430, E3 +6269.387}
SPL {X  -160.000, Y  +418.225, Z    +0.000, E1   +21.425, E3 +6288.069}
SPL {X  -160.000, Y  +414.956, Z    +0.000, E1   +21.424, E3 +6305.749}
SPL {X  -160.000, Y  +411.834, Z    +0.000, E1   +21.420, E3 +6322.667}
SPL {X  -160.000, Y  +408.570, Z    +0.000, E1   +21.432, E3 +6340.277}
SPL {X  -160.000, Y  +405.237, Z    +0.000, E1   +21.432, E3 +6358.305}
SPL {X  -160.000, Y  +402.004, Z    +0.000, E1   +21.424, E3 +6375.880}
SPL {X  -160.000, Y  +398.626, Z    +0.000, E1   +21.425, E3 +6394.186}
SPL {X  -160.000, Y  +395.405, Z    +0.000, E1   +21.422, E3 +6411.604}
SPL {X  -160.000, Y  +392.641, Z    +0.000, E1   +21.407, E3 +6426.602}
SPL {X  -159.989, Y  +390.129, Z    +0.000, E1   +21.406, E3 +6440.243}
SPL {X  -159.932, Y  +387.337, Z    +0.000, E1   +21.403, E3 +6455.439}
SPL {X  -159.823, Y  +384.478, Z    +0.000, E1   +21.379, E3 +6471.102}
SPL {X  -159.660, Y  +381.581, Z    +0.000, E1   +21.363, E3 +6486.990}
SPL {X  -159.452, Y  +378.773, Z    +0.000, E1   +21.330, E3 +6502.437}
SPL {X  -159.222, Y  +376.244, Z    +0.000, E1   +21.297, E3 +6516.399}
SPL {X  -158.814, Y  +372.556, Z    +0.000, E1   +21.316, E3 +6536.666}
SPL {X  -158.301, Y  +368.743, Z    +0.000, E1   +21.199, E3 +6557.988}
SPL {X  -157.981, Y  +366.660, Z    +0.000, E1   +19.986, E3 +6580.956}
ENDSPLINE

SPLINE
SPL {X  -158.491, Y  +370.077, Z    +0.000, E1   +15.910, E3 +6605.969}
SPL {X  -159.771, Y  +383.450, Z    +0.000, E1    +6.314, E3 +6629.124}
SPL {X  -160.000, Y  +392.463, Z    +0.000, E1    +0.112, E3 +6635.631}
SPL {X  -160.000, Y  +399.874, Z    +0.000, E1    -5.508, E3 +6640.133}
SPL {X  -160.000, Y  +411.622, Z    +0.000, E1   -13.815, E3 +6652.253}
SPL {X  -160.000, Y  +419.836, Z    +0.000, E1   -18.198, E3 +6667.427}
SPL {X  -160.000, Y  +430.523, Z    +0.000, E1   -21.710, E3 +6697.627}
SPL {X  -160.000, Y  +433.426, Z    +0.000, E1   -21.735, E3 +6713.042}
SPL {X  -160.000, Y  +436.131, Z    +0.000, E1   -21.710, E3 +6727.517}
SPL {X  -160.000, Y  +439.046, Z    +0.000, E1   -21.732, E3 +6743.010}
SPL {X  -160.000, Y  +442.009, Z    +0.000, E1   -21.719, E3 +6758.832}
SPL {X  -160.000, Y  +444.891, Z    +0.000, E1   -21.724, E3 +6774.188}
SPL {X  -160.000, Y  +449.017, Z    +0.000, E1   -21.792, E3 +6795.979}
SPL {X  -160.000, Y  +452.864, Z    +0.000, E1   -21.730, E3 +6816.597}
SPL {X  -160.000, Y  +455.470, Z    +0.000, E1   -21.722, E3 +6830.486}
SPL {X  -160.000, Y  +458.295, Z    +0.000, E1   -21.738, E3 +6845.507}
SPL {X  -160.000, Y  +461.133, Z    +0.000, E1   -21.720, E3 +6860.690}
SPL {X  -160.000, Y  +464.458, Z    +0.000, E1   -21.770, E3 +6878.208}
SPL {X  -160.000, Y  +468.250, Z    +0.000, E1   -21.764, E3 +6898.361}
SPL {X  -160.000, Y  +472.226, Z    +0.000, E1   -21.782, E3 +6919.520}
SPL {X  -160.000, Y  +476.333, Z    +0.000, E1   -21.767, E3 +6941.434}
SPL {X  -160.000, Y  +480.244, Z    +0.000, E1   -21.765, E3 +6962.299}
SPL {X  -160.000, Y  +484.301, Z    +0.000, E1   -21.775, E3 +6983.827}
SPL {X  -160.000, Y  +488.201, Z    +0.000, E1   -21.768, E3 +7004.587}
SPL {X  -160.000, Y  +492.394, Z    +0.000, E1   -21.802, E3 +7026.761}
SPL {X  -160.000, Y  +496.781, Z    +0.000, E1   -21.798, E3 +7050.073}
SPL {X  -160.000, Y  +501.083, Z    +0.000, E1   -21.796, E3 +7073.003}
SPL {X  -160.000, Y  +504.917, Z    +0.000, E1   -21.764, E3 +7093.507}
SPL {X  -160.000, Y  +508.886, Z    +0.000, E1   -21.791, E3 +7114.593}
SPL {X  -160.000, Y  +513.057, Z    +0.000, E1   -21.767, E3 +7136.901}
SPL {X  -160.000, Y  +517.221, Z    +0.000, E1   -21.778, E3 +7159.054}
SPL {X  -160.000, Y  +521.677, Z    +0.000, E1   -21.781, E3 +7182.815}
SPL {X  -160.000, Y  +525.729, Z    +0.000, E1   -21.753, E3 +7204.454}
SPL {X  -160.000, Y  +529.456, Z    +0.000, E1   -21.766, E3 +7224.234}
SPL {X  -160.000, Y  +533.608, Z    +0.000, E1   -21.776, E3 +7246.364}
SPL {X  -160.000, Y  +538.227, Z    +0.000, E1   -21.794, E3 +7270.896}
SPL {X  -160.000, Y  +542.483, Z    +0.000, E1   -21.764, E3 +7293.622}
SPL {X  -160.000, Y  +546.194, Z    +0.000, E1   -21.754, E3 +7313.438}
SPL {X  -160.000, Y  +550.131, Z    +0.000, E1   -21.771, E3 +7334.374}
SPL {X  -160.000, Y  +554.462, Z    +0.000, E1   -21.777, E3 +7357.428}
SPL {X  -160.000, Y  +558.542, Z    +0.000, E1   -21.758, E3 +7379.200}
SPL {X  -160.000, Y  +562.615, Z    +0.000, E1   -21.776, E3 +7400.856}
SPL {X  -160.000, Y  +566.764, Z    +0.000, E1   -21.764, E3 +7422.981}
SPL {X  -160.000, Y  +570.657, Z    +0.000, E1   -21.758, E3 +7443.728}
SPL {X  -160.000, Y  +574.688, Z    +0.000, E1   -21.771, E3 +7465.171}
SPL {X  -160.000, Y  +578.864, Z    +0.000, E1   -21.770, E3 +7487.422}
SPL {X  -160.000, Y  +582.807, Z    +0.000, E1   -21.754, E3 +7508.476}
SPL {X  -160.000, Y  +586.993, Z    +0.000, E1   -21.779, E3 +7530.712}
SPL {X  -160.000, Y  +591.368, Z    +0.000, E1   -21.775, E3 +7553.999}
SPL {X  -160.000, Y  +595.703, Z    +0.000, E1   -21.775, E3 +7577.108}
SPL {X  -160.000, Y  +599.558, Z    +0.000, E1   -21.748, E3 +7597.686}
SPL {X  -160.000, Y  +603.126, Z    +0.000, E1   -21.757, E3 +7616.665}
SPL {X  -160.000, Y  +607.107, Z    +0.000, E1   -21.766, E3 +7637.891}
SPL {X  -160.000, Y  +611.246, Z    +0.000, E1   -21.760, E3 +7659.964}
SPL {X  -160.000, Y  +615.151, Z    +0.000, E1   -21.752, E3 +7680.777}
SPL {X  -160.000, Y  +618.728, Z    +0.000, E1   -21.747, E3 +7699.839}
SPL {X  -160.000, Y  +622.318, Z    +0.000, E1   -21.753, E3 +7718.954}
SPL {X  -160.000, Y  +625.877, Z    +0.000, E1   -21.745, E3 +7737.932}
SPL {X  -160.000, Y  +629.892, Z    +0.000, E1   -21.777, E3 +7759.256}
SPL {X  -160.000, Y  +634.024, Z    +0.000, E1   -21.756, E3 +7781.306}
SPL {X  -160.000, Y  +637.661, Z    +0.000, E1   -21.748, E3 +7800.697}
SPL {X  -160.000, Y  +641.244, Z    +0.000, E1   -21.752, E3 +7819.768}
SPL {X  -160.000, Y  +645.120, Z    +0.000, E1   -21.762, E3 +7840.400}
SPL {X  -160.000, Y  +649.214, Z    +0.000, E1   -21.766, E3 +7862.188}
SPL {X  -160.000, Y  +653.188, Z    +0.000, E1   -21.771, E3 +7883.251}
SPL {X  -160.000, Y  +656.905, Z    +0.000, E1   -21.769, E3 +7903.026}
SPL {X  -160.000, Y  +660.685, Z    +0.000, E1   -21.769, E3 +7923.194}
SPL {X  -160.000, Y  +664.985, Z    +0.000, E1   -21.790, E3 +7946.047}
SPL {X  -159.993, Y  +669.170, Z    +0.000, E1   -21.763, E3 +7968.405}
SPL {X  -159.916, Y  +672.869, Z    +0.000, E1   -21.755, E3 +7988.150}
SPL {X  -159.752, Y  +676.610, Z    +0.000, E1   -21.740, E3 +8008.225}
SPL {X  -159.478, Y  +680.618, Z    +0.000, E1   -21.719, E3 +8029.824}
SPL {X  -159.108, Y  +684.576, Z    +0.000, E1   -21.664, E3 +8051.294}
SPL {X  -158.638, Y  +688.530, Z    +0.000, E1   -21.617, E3 +8072.815}
SPL {X  -158.097, Y  +692.303, Z    +0.000, E1   -21.529, E3 +8093.533}
ENDSPLINE

SPLINE
SPL {X  -158.264, Y  +691.203, Z    +0.000, E1   -17.264, E3 +8130.278}
SPL {X  -159.000, Y  +685.560, Z    +0.000, E1   -12.398, E3 +8151.454}
SPL {X  -159.924, Y  +672.625, Z    +0.000, E1    -3.689, E3 +8166.471}
SPL {X  -160.000, Y  +663.203, Z    +0.000, E1    +3.155, E3 +8173.125}
SPL {X  -160.000, Y  +652.103, Z    +0.000, E1   +11.247, E3 +8184.795}
SPL {X  -160.000, Y  +641.822, Z    +0.000, E1   +17.059, E3 +8204.169}
SPL {X  -160.000, Y  +631.293, Z    +0.000, E1   +20.354, E3 +8238.049}
SPL {X  -160.000, Y  +627.542, Z    +0.000, E1   +20.380, E3 +8259.456}
SPL {X  -160.000, Y  +623.532, Z    +0.000, E1   +20.378, E3 +8282.421}
SPL {X  -160.000, Y  +619.329, Z    +0.000, E1   +20.391, E3 +8306.459}
SPL {X  -160.000, Y  +614.967, Z    +0.000, E1   +20.392, E3 +8331.439}
SPL {X  -160.000, Y  +611.206, Z    +0.000, E1   +20.351, E3 +8353.111}
SPL {X  -160.000, Y  +607.824, Z    +0.000, E1   +20.354, E3 +8372.531}
SPL {X  -160.000, Y  +603.899, Z    +0.000, E1   +20.373, E3 +8394.981}
SPL {X  -160.000, Y  +599.617, Z    +0.000, E1   +20.384, E3 +8419.475}
SPL {X  -160.000, Y  +595.532, Z    +0.000, E1   +20.373, E3 +8442.836}
SPL {X  -160.000, Y  +591.705, Z    +0.000, E1   +20.373, E3 +8464.760}
SPL {X  -160.000, Y  +588.037, Z    +0.000, E1   +20.359, E3 +8485.847}
SPL {X  -160.000, Y  +584.320, Z    +0.000, E1   +20.364, E3 +8507.149}
SPL {X  -160.000, Y  +580.616, Z    +0.000, E1   +20.357, E3 +8528.376}
SPL {X  -160.000, Y  +577.083, Z    +0.000, E1   +20.358, E3 +8548.624}
SPL {X  -160.000, Y  +573.158, Z    +0.000, E1   +20.377, E3 +8571.076}
SPL {X  -160.000, Y  +568.802, Z    +0.000, E1   +20.385, E3 +8596.028}
SPL {X  -160.000, Y  +564.937, Z    +0.000, E1   +20.350, E3 +8618.249}
SPL {X  -160.000, Y  +561.213, Z    +0.000, E1   +20.372, E3 +8639.535}
SPL {X  -160.000, Y  +557.320, Z    +0.000, E1   +20.363, E3 +8661.862}
SPL {X  -160.000, Y  +553.712, Z    +0.000, E1   +20.355, E3 +8682.561}
SPL {X  -160.000, Y  +550.040, Z    +0.000, E1   +20.360, E3 +8703.600}
SPL {X  -160.000, Y  +546.180, Z    +0.000, E1   +20.370, E3 +8725.655}
SPL {X  -160.000, Y  +542.032, Z    +0.000, E1   +20.384, E3 +8749.394}
SPL {X  -160.000, Y  +537.870, Z    +0.000, E1   +20.372, E3 +8773.270}
SPL {X  -160.000, Y  +534.086, Z    +0.000, E1   +20.356, E3 +8795.024}
SPL {X  -160.000, Y  +530.164, Z    +0.000, E1   +20.382, E3 +8817.373}
SPL {X  -160.000, Y  +527.505, Z    +0.000, E1   +20.318, E3 +8832.747}
SPL {X  -160.000, Y  +511.620, Z    +0.000, E1   +28.365, E3 +8843.210}
SPL {X  -160.000, Y  +507.906, Z    +0.000, E1   +28.152, E3 +8859.605}
SPL {X  -160.000, Y  +506.085, Z    +0.000, E1   +26.146, E3 +8882.065}
SPL {X  -160.000, Y  +504.342, Z    +0.000, E1   +24.109, E3 +8905.580}
SPL {X  -160.000, Y  +503.002, Z    +0.000, E1   +22.325, E3 +8926.585}
SPL {X  -160.000, Y  +500.783, Z    +0.000, E1   +21.421, E3 +8946.175}
SPL {X  -160.000, Y  +497.229, Z    +0.000, E1   +21.403, E3 +8965.483}
SPL {X  -160.000, Y  +493.901, Z    +0.000, E1   +21.409, E3 +8983.502}
SPL {X  -160.000, Y  +490.791, Z    +0.000, E1   +21.400, E3 +9000.375}
SPL {X  -160.000, Y  +487.647, Z    +0.000, E1   +21.401, E3 +9017.421}
SPL {X  -160.000, Y  +484.273, Z    +0.000, E1   +21.408, E3 +9035.701}
SPL {X  -160.000, Y  +481.093, Z    +0.000, E1   +21.389, E3 +9053.010}
SPL {X  -160.000, Y  +478.021, Z    +0.000, E1   +21.401, E3 +9069.616}
SPL {X  -160.000, Y  +474.639, Z    +0.000, E1   +21.410, E3 +9087.908}
SPL {X  -160.000, Y  +471.343, Z    +0.000, E1   +21.399, E3 +9105.810}
SPL {X  -160.000, Y  +468.133, Z    +0.000, E1   +21.402, E3 +9123.201}
SPL {X  -160.000, Y  +464.638, Z    +0.000, E1   +21.421, E3 +9142.050}
SPL {X  -160.000, Y  +461.045, Z    +0.000, E1   +21.424, E3 +9161.464}
SPL {X  -160.000, Y  +457.606, Z    +0.000, E1   +21.413, E3 +9180.174}
SPL {X  -160.000, Y  +454.417, Z    +0.000, E1   +21.401, E3 +9197.483}
SPL {X  -160.000, Y  +451.425, Z    +0.000, E1   +21.404, E3 +9213.704}
SPL {X  -160.000, Y  +448.039, Z    +0.000, E1   +21.417, E3 +9231.997}
SPL {X  -160.000, Y  +444.787, Z    +0.000, E1   +21.414, E3 +9249.553}
SPL {X  -160.000, Y  +441.637, Z    +0.000, E1   +21.431, E3 +9266.531}
SPL {X  -160.000, Y  +438.199, Z    +0.000, E1   +21.432, E3 +9285.134}
SPL {X  -160.000, Y  +434.875, Z    +0.000, E1   +21.424, E3 +9303.174}
SPL {X  -160.000, Y  +431.689, Z    +0.000, E1   +21.423, E3 +9320.423}
SPL {X  -160.000, Y  +428.451, Z    +0.000, E1   +21.430, E3 +9337.902}
SPL {X  -160.000, Y  +425.120, Z    +0.000, E1   +21.430, E3 +9355.967}
SPL {X  -160.000, Y  +421.671, Z    +0.000, E1   +21.430, E3 +9374.650}
SPL {X  -160.000, Y  +418.225, Z    +0.000, E1   +21.425, E3 +9393.332}
SPL {X  -160.000, Y  +414.956, Z    +0.000, E1   +21.424, E3 +9411.013}
SPL {X  -160.000, Y  +411.834, Z    +0.000, E1   +21.420, E3 +9427.931}
SPL {X  -160.000, Y  +408.570, Z    +0.000, E1   +21.432, E3 +9445.540}
SPL {X  -160.000, Y  +405.237, Z    +0.000, E1   +21.432, E3 +9463.568}
SPL {X  -160.000, Y  +402.004, Z    +0.000, E1   +21.424, E3 +9481.144}
SPL {X  -160.000, Y  +398.626, Z    +0.000, E1   +21.425, E3 +9499.450}
SPL {X  -160.000, Y  +395.405, Z    +0.000, E1   +21.422, E3 +9516.867}
SPL {X  -160.000, Y  +392.641, Z    +0.000, E1   +21.407, E3 +9531.866}
SPL {X  -159.989, Y  +390.129, Z    +0.000, E1   +21.406, E3 +9545.507}
SPL {X  -159.932, Y  +387.337, Z    +0.000, E1   +21.403, E3 +9560.702}
SPL {X  -159.823, Y  +384.478, Z    +0.000, E1   +21.379, E3 +9576.366}
SPL {X  -159.660, Y  +381.581, Z    +0.000, E1   +21.363, E3 +9592.254}
SPL {X  -159.452, Y  +378.773, Z    +0.000, E1   +21.330, E3 +9607.700}
SPL {X  -159.222, Y  +376.244, Z    +0.000, E1   +21.297, E3 +9621.663}
SPL {X  -158.814, Y  +372.556, Z    +0.000, E1   +21.316, E3 +9641.930}
SPL {X  -158.301, Y  +368.743, Z    +0.000, E1   +21.199, E3 +9663.252}
SPL {X  -157.981, Y  +366.660, Z    +0.000, E1   +19.986, E3 +9686.219}
ENDSPLINE

SPLINE
SPL {X  -158.491, Y  +370.077, Z    +0.000, E1   +15.910, E3 +9711.232}
SPL {X  -159.771, Y  +383.450, Z    +0.000, E1    +6.314, E3 +9734.388}
SPL {X  -160.000, Y  +392.463, Z    +0.000, E1    +0.112, E3 +9740.894}
SPL {X  -160.000, Y  +399.874, Z    +0.000, E1    -5.508, E3 +9745.397}
SPL {X  -160.000, Y  +411.622, Z    +0.000, E1   -13.815, E3 +9757.517}
SPL {X  -160.000, Y  +419.836, Z    +0.000, E1   -18.198, E3 +9772.691}
SPL {X  -160.000, Y  +430.523, Z    +0.000, E1   -21.710, E3 +9802.891}
SPL {X  -160.000, Y  +433.426, Z    +0.000, E1   -21.735, E3 +9818.305}
SPL {X  -160.000, Y  +436.131, Z    +0.000, E1   -21.710, E3 +9832.780}
SPL {X  -160.000, Y  +439.046, Z    +0.000, E1   -21.732, E3 +9848.273}
SPL {X  -160.000, Y  +442.009, Z    +0.000, E1   -21.719, E3 +9864.095}
SPL {X  -160.000, Y  +444.891, Z    +0.000, E1   -21.724, E3 +9879.451}
SPL {X  -160.000, Y  +449.017, Z    +0.000, E1   -21.792, E3 +9901.243}
SPL {X  -160.000, Y  +452.864, Z    +0.000, E1   -21.730, E3 +9921.860}
SPL {X  -160.000, Y  +455.470, Z    +0.000, E1   -21.722, E3 +9935.749}
SPL {X  -160.000, Y  +458.295, Z    +0.000, E1   -21.738, E3 +9950.770}
SPL {X  -160.000, Y  +461.133, Z    +0.000, E1   -21.720, E3 +9965.953}
SPL {X  -160.000, Y  +464.458, Z    +0.000, E1   -21.770, E3 +9983.472}
SPL {X  -160.000, Y  +468.250, Z    +0.000, E1   -21.764, E3 +10003.625}
SPL {X  -160.000, Y  +472.226, Z    +0.000, E1   -21.782, E3 +10024.783}
SPL {X  -160.000, Y  +476.333, Z    +0.000, E1   -21.767, E3 +10046.698}
SPL {X  -160.000, Y  +480.244, Z    +0.000, E1   -21.765, E3 +10067.562}
SPL {X  -160.000, Y  +484.301, Z    +0.000, E1   -21.775, E3 +10089.091}
SPL {X  -160.000, Y  +488.201, Z    +0.000, E1   -21.768, E3 +10109.851}
SPL {X  -160.000, Y  +492.394, Z    +0.000, E1   -21.802, E3 +10132.025}
SPL {X  -160.000, Y  +496.781, Z    +0.000, E1   -21.798, E3 +10155.336}
SPL {X  -160.000, Y  +501.083, Z    +0.000, E1   -21.796, E3 +10178.266}
SPL {X  -160.000, Y  +504.917, Z    +0.000, E1   -21.764, E3 +10198.771}
SPL {X  -160.000, Y  +508.886, Z    +0.000, E1   -21.791, E3 +10219.857}
SPL {X  -160.000, Y  +513.057, Z    +0.000, E1   -21.767, E3 +10242.164}
SPL {X  -160.000, Y  +517.221, Z    +0.000, E1   -21.778, E3 +10264.317}
SPL {X  -160.000, Y  +521.677, Z    +0.000, E1   -21.781, E3 +10288.078}
SPL {X  -160.000, Y  +525.729, Z    +0.000, E1   -21.753, E3 +10309.718}
SPL {X  -160.000, Y  +529.456, Z    +0.000, E1   -21.766, E3 +10329.497}
SPL {X  -160.000, Y  +533.608, Z    +0.000, E1   -21.776, E3 +10351.627}
SPL {X  -160.000, Y  +538.227, Z    +0.000, E1   -21.794, E3 +10376.160}
SPL {X  -160.000, Y  +542.483, Z    +0.000, E1   -21.764, E3 +10398.885}
SPL {X  -160.000, Y  +546.194, Z    +0.000, E1   -21.754, E3 +10418.702}
SPL {X  -160.000, Y  +550.131, Z    +0.000, E1   -21.771, E3 +10439.637}
SPL {X  -160.000, Y  +554.462, Z    +0.000, E1   -21.777, E3 +10462.691}
SPL {X  -160.000, Y  +558.542, Z    +0.000, E1   -21.758, E3 +10484.464}
SPL {X  -160.000, Y  +562.615, Z    +0.000, E1   -21.776, E3 +10506.120}
SPL {X  -160.000, Y  +566.764, Z    +0.000, E1   -21.764, E3 +10528.245}
SPL {X  -160.000, Y  +570.657, Z    +0.000, E1   -21.758, E3 +10548.992}
SPL {X  -160.000, Y  +574.688, Z    +0.000, E1   -21.771, E3 +10570.435}
SPL {X  -160.000, Y  +578.864, Z    +0.000, E1   -21.770, E3 +10592.686}
SPL {X  -160.000, Y  +582.807, Z    +0.000, E1   -21.754, E3 +10613.740}
SPL {X  -160.000, Y  +586.993, Z    +0.000, E1   -21.779, E3 +10635.975}
SPL {X  -160.000, Y  +591.368, Z    +0.000, E1   -21.775, E3 +10659.262}
SPL {X  -160.000, Y  +595.703, Z    +0.000, E1   -21.775, E3 +10682.372}
SPL {X  -160.000, Y  +599.558, Z    +0.000, E1   -21.748, E3 +10702.949}
SPL {X  -160.000, Y  +603.126, Z    +0.000, E1   -21.757, E3 +10721.929}
SPL {X  -160.000, Y  +607.107, Z    +0.000, E1   -21.766, E3 +10743.154}
SPL {X  -160.000, Y  +611.246, Z    +0.000, E1   -21.760, E3 +10765.227}
SPL {X  -160.000, Y  +615.151, Z    +0.000, E1   -21.752, E3 +10786.041}
SPL {X  -160.000, Y  +618.728, Z    +0.000, E1   -21.747, E3 +10805.103}
SPL {X  -160.000, Y  +622.318, Z    +0.000, E1   -21.753, E3 +10824.217}
SPL {X  -160.000, Y  +625.877, Z    +0.000, E1   -21.745, E3 +10843.196}
SPL {X  -160.000, Y  +629.892, Z    +0.000, E1   -21.777, E3 +10864.520}
SPL {X  -160.000, Y  +634.024, Z    +0.000, E1   -21.756, E3 +10886.570}
SPL {X  -160.000, Y  +637.661, Z    +0.000, E1   -21.748, E3 +10905.961}
SPL {X  -160.000, Y  +641.244, Z    +0.000, E1   -21.752, E3 +10925.031}
SPL {X  -160.000, Y  +645.120, Z    +0.000, E1   -21.762, E3 +10945.664}
SPL {X  -160.000, Y  +649.214, Z    +0.000, E1   -21.766, E3 +10967.452}
SPL {X  -160.000, Y  +653.188, Z    +0.000, E1   -21.771, E3 +10988.514}
SPL {X  -160.000, Y  +656.905, Z    +0.000, E1   -21.769, E3 +11008.290}
SPL {X  -160.000, Y  +660.685, Z    +0.000, E1   -21.769, E3 +11028.458}
SPL {X  -160.000, Y  +664.985, Z    +0.000, E1   -21.790, E3 +11051.310}
SPL {X  -159.993, Y  +669.170, Z    +0.000, E1   -21.763, E3 +11073.669}
SPL {X  -159.916, Y  +672.869, Z    +0.000, E1   -21.755, E3 +11093.414}
SPL {X  -159.752, Y  +676.610, Z    +0.000, E1   -21.740, E3 +11113.489}
SPL {X  -159.478, Y  +680.618, Z    +0.000, E1   -21.719, E3 +11135.088}
SPL {X  -159.108, Y  +684.576, Z    +0.000, E1   -21.664, E3 +11156.557}
SPL {X  -158.638, Y  +688.530, Z    +0.000, E1   -21.617, E3 +11178.079}
SPL {X  -158.097, Y  +692.303, Z    +0.000, E1   -21.529, E3 +11198.796}
ENDSPLINE

SPLINE
SPL {X  -158.264, Y  +691.203, Z    +0.000, E1   -17.264, E3 +11235.542}
SPL {X  -159.000, Y  +685.560, Z    +0.000, E1   -12.398, E3 +11256.717}
SPL {X  -159.924, Y  +672.625, Z    +0.000, E1    -3.689, E3 +11271.734}
SPL {X  -160.000, Y  +663.203, Z    +0.000, E1    +3.155, E3 +11278.389}
SPL {X  -160.000, Y  +652.103, Z    +0.000, E1   +11.247, E3 +11290.059}
SPL {X  -160.000, Y  +641.822, Z    +0.000, E1   +17.059, E3 +11309.433}
SPL {X  -160.000, Y  +631.293, Z    +0.000, E1   +20.354, E3 +11343.312}
SPL {X  -160.000, Y  +627.542, Z    +0.000, E1   +20.380, E3 +11364.719}
SPL {X  -160.000, Y  +623.532, Z    +0.000, E1   +20.378, E3 +11387.685}
SPL {X  -160.000, Y  +619.329, Z    +0.000, E1   +20.391, E3 +11411.722}
SPL {X  -160.000, Y  +614.967, Z    +0.000, E1   +20.392, E3 +11436.702}
SPL {X  -160.000, Y  +611.206, Z    +0.000, E1   +20.351, E3 +11458.374}
SPL {X  -160.000, Y  +607.824, Z    +0.000, E1   +20.354, E3 +11477.795}
SPL {X  -160.000, Y  +603.899, Z    +0.000, E1   +20.373, E3 +11500.245}
SPL {X  -160.000, Y  +599.617, Z    +0.000, E1   +20.384, E3 +11524.739}
SPL {X  -160.000, Y  +595.532, Z    +0.000, E1   +20.373, E3 +11548.099}
SPL {X  -160.000, Y  +591.705, Z    +0.000, E1   +20.373, E3 +11570.024}
SPL {X  -160.000, Y  +588.037, Z    +0.000, E1   +20.359, E3 +11591.111}
SPL {X  -160.000, Y  +584.320, Z    +0.000, E1   +20.364, E3 +11612.412}
SPL {X  -160.000, Y  +580.616, Z    +0.000, E1   +20.357, E3 +11633.639}
SPL {X  -160.000, Y  +577.083, Z    +0.000, E1   +20.358, E3 +11653.888}
SPL {X  -160.000, Y  +573.158, Z    +0.000, E1   +20.377, E3 +11676.340}
SPL {X  -160.000, Y  +568.802, Z    +0.000, E1   +20.385, E3 +11701.292}
SPL {X  -160.000, Y  +564.937, Z    +0.000, E1   +20.350, E3 +11723.512}
SPL {X  -160.000, Y  +561.213, Z    +0.000, E1   +20.372, E3 +11744.799}
SPL {X  -160.000, Y  +557.320, Z    +0.000, E1   +20.363, E3 +11767.126}
SPL {X  -160.000, Y  +553.712, Z    +0.000, E1   +20.355, E3 +11787.825}
SPL {X  -160.000, Y  +550.040, Z    +0.000, E1   +20.360, E3 +11808.863}
SPL {X  -160.000, Y  +546.180, Z    +0.000, E1   +20.370, E3 +11830.919}
SPL {X  -160.000, Y  +542.032, Z    +0.000, E1   +20.384, E3 +11854.658}
SPL {X  -160.000, Y  +537.870, Z    +0.000, E1   +20.372, E3 +11878.533}
SPL {X  -160.000, Y  +534.086, Z    +0.000, E1   +20.356, E3 +11900.287}
SPL {X  -160.000, Y  +530.164, Z    +0.000, E1   +20.382, E3 +11922.637}
SPL {X  -160.000, Y  +527.505, Z    +0.000, E1   +20.318, E3 +11938.011}
SPL {X  -160.000, Y  +511.620, Z    +0.000, E1   +28.365, E3 +11948.474}
SPL {X  -160.000, Y  +507.906, Z    +0.000, E1   +28.152, E3 +11964.869}
SPL {X  -160.000, Y  +506.085, Z    +0.000, E1   +26.146, E3 +11987.328}
SPL {X  -160.000, Y  +504.342, Z    +0.000, E1   +24.109, E3 +12010.843}
SPL {X  -160.000, Y  +503.002, Z    +0.000, E1   +22.325, E3 +12031.849}
SPL {X  -160.000, Y  +500.783, Z    +0.000, E1   +21.421, E3 +12051.438}
SPL {X  -160.000, Y  +497.229, Z    +0.000, E1   +21.403, E3 +12070.746}
SPL {X  -160.000, Y  +493.901, Z    +0.000, E1   +21.409, E3 +12088.765}
SPL {X  -160.000, Y  +490.791, Z    +0.000, E1   +21.400, E3 +12105.638}
SPL {X  -160.000, Y  +487.647, Z    +0.000, E1   +21.401, E3 +12122.684}
SPL {X  -160.000, Y  +484.273, Z    +0.000, E1   +21.408, E3 +12140.964}
SPL {X  -160.000, Y  +481.093, Z    +0.000, E1   +21.389, E3 +12158.273}
SPL {X  -160.000, Y  +478.021, Z    +0.000, E1   +21.401, E3 +12174.880}
SPL {X  -160.000, Y  +474.639, Z    +0.000, E1   +21.410, E3 +12193.171}
SPL {X  -160.000, Y  +471.343, Z    +0.000, E1   +21.399, E3 +12211.073}
SPL {X  -160.000, Y  +468.133, Z    +0.000, E1   +21.402, E3 +12228.465}
SPL {X  -160.000, Y  +464.638, Z    +0.000, E1   +21.421, E3 +12247.314}
SPL {X  -160.000, Y  +461.045, Z    +0.000, E1   +21.424, E3 +12266.728}
SPL {X  -160.000, Y  +457.606, Z    +0.000, E1   +21.413, E3 +12285.438}
SPL {X  -160.000, Y  +454.417, Z    +0.000, E1   +21.401, E3 +12302.746}
SPL {X  -160.000, Y  +451.425, Z    +0.000, E1   +21.404, E3 +12318.968}
SPL {X  -160.000, Y  +448.039, Z    +0.000, E1   +21.417, E3 +12337.261}
SPL {X  -160.000, Y  +444.787, Z    +0.000, E1   +21.414, E3 +12354.816}
SPL {X  -160.000, Y  +441.637, Z    +0.000, E1   +21.431, E3 +12371.794}
SPL {X  -160.000, Y  +438.199, Z    +0.000, E1   +21.432, E3 +12390.398}
SPL {X  -160.000, Y  +434.875, Z    +0.000, E1   +21.424, E3 +12408.438}
SPL {X  -160.000, Y  +431.689, Z    +0.000, E1   +21.423, E3 +12425.686}
SPL {X  -160.000, Y  +428.451, Z    +0.000, E1   +21.430, E3 +12443.166}
SPL {X  -160.000, Y  +425.120, Z    +0.000, E1   +21.430, E3 +12461.230}
SPL {X  -160.000, Y  +421.671, Z    +0.000, E1   +21.430, E3 +12479.914}
SPL {X  -160.000, Y  +418.225, Z    +0.000, E1   +21.425, E3 +12498.596}
SPL {X  -160.000, Y  +414.956, Z    +0.000, E1   +21.424, E3 +12516.276}
SPL {X  -160.000, Y  +411.834, Z    +0.000, E1   +21.420, E3 +12533.195}
SPL {X  -160.000, Y  +408.570, Z    +0.000, E1   +21.432, E3 +12550.804}
SPL {X  -160.000, Y  +405.237, Z    +0.000, E1   +21.432, E3 +12568.832}
SPL {X  -160.000, Y  +402.004, Z    +0.000, E1   +21.424, E3 +12586.407}
SPL {X  -160.000, Y  +398.626, Z    +0.000, E1   +21.425, E3 +12604.713}
SPL {X  -160.000, Y  +395.405, Z    +0.000, E1   +21.422, E3 +12622.131}
SPL {X  -160.000, Y  +392.641, Z    +0.000, E1   +21.407, E3 +12637.129}
SPL {X  -159.989, Y  +390.129, Z    +0.000, E1   +21.406, E3 +12650.770}
SPL {X  -159.932, Y  +387.337, Z    +0.000, E1   +21.403, E3 +12665.966}
SPL {X  -159.823, Y  +384.478, Z    +0.000, E1   +21.379, E3 +12681.629}
SPL {X  -159.660, Y  +381.581, Z    +0.000, E1   +21.363, E3 +12697.517}
SPL {X  -159.452, Y  +378.773, Z    +0.000, E1   +21.330, E3 +12712.964}
SPL {X  -159.222, Y  +376.244, Z    +0.000, E1   +21.297, E3 +12726.926}
SPL {X  -158.814, Y  +372.556, Z    +0.000, E1   +21.316, E3 +12747.193}
SPL {X  -158.301, Y  +368.743, Z    +0.000, E1   +21.199, E3 +12768.515}
SPL {X  -157.981, Y  +366.660, Z    +0.000, E1   +19.986, E3 +12791.483}
ENDSPLINE

SPLINE
SPL {X  -158.491, Y  +370.077, Z    +0.000, E1   +15.910, E3 +12816.496}
SPL {X  -159.771, Y  +383.450, Z    +0.000, E1    +6.314, E3 +12839.651}
SPL {X  -160.000, Y  +392.463, Z    +0.000, E1    +0.112, E3 +12846.158}
SPL {X  -160.000, Y  +399.874, Z    +0.000, E1    -5.508, E3 +12850.660}
SPL {X  -160.000, Y  +411.622, Z    +0.000, E1   -13.815, E3 +12862.780}
SPL {X  -160.000, Y  +419.836, Z    +0.000, E1   -18.198, E3 +12877.954}
SPL {X  -160.000, Y  +430.523, Z    +0.000, E1   -21.710, E3 +12908.154}
SPL {X  -160.000, Y  +433.426, Z    +0.000, E1   -21.735, E3 +12923.569}
SPL {X  -160.000, Y  +436.131, Z    +0.000, E1   -21.710, E3 +12938.044}
SPL {X  -160.000, Y  +439.046, Z    +0.000, E1   -21.732, E3 +12953.537}
SPL {X  -160.000, Y  +442.009, Z    +0.000, E1   -21.719, E3 +12969.359}
SPL {X  -160.000, Y  +444.891, Z    +0.000, E1   -21.724, E3 +12984.715}
SPL {X  -160.000, Y  +449.017, Z    +0.000, E1   -21.792, E3 +13006.506}
SPL {X  -160.000, Y  +452.864, Z    +0.000, E1   -21.730, E3 +13027.124}
SPL {X  -160.000, Y  +455.470, Z    +0.000, E1   -21.722, E3 +13041.013}
SPL {X  -160.000, Y  +458.295, Z    +0.000, E1   -21.738, E3 +13056.034}
SPL {X  -160.000, Y  +461.133, Z    +0.000, E1   -21.720, E3 +13071.217}
SPL {X  -160.000, Y  +464.458, Z    +0.000, E1   -21.770, E3 +13088.735}
SPL {X  -160.000, Y  +468.250, Z    +0.000, E1   -21.764, E3 +13108.888}
SPL {X  -160.000, Y  +472.226, Z    +0.000, E1   -21.782, E3 +13130.047}
SPL {X  -160.000, Y  +476.333, Z    +0.000, E1   -21.767, E3 +13151.961}
SPL {X  -160.000, Y  +480.244, Z    +0.000, E1   -21.765, E3 +13172.826}
SPL {X  -160.000, Y  +484.301, Z    +0.000, E1   -21.775, E3 +13194.354}
SPL {X  -160.000, Y  +488.201, Z    +0.000, E1   -21.768, E3 +13215.114}
SPL {X  -160.000, Y  +492.394, Z    +0.000, E1   -21.802, E3 +13237.289}
SPL {X  -160.000, Y  +496.781, Z    +0.000, E1   -21.798, E3 +13260.600}
SPL {X  -160.000, Y  +501.083, Z    +0.000, E1   -21.796, E3 +13283.530}
SPL {X  -160.000, Y  +504.917, Z    +0.000, E1   -21.764, E3 +13304.034}
SPL {X  -160.000, Y  +508.886, Z    +0.000, E1   -21.791, E3 +13325.120}
SPL {X  -160.000, Y  +513.057, Z    +0.000, E1   -21.767, E3 +13347.428}
SPL {X  -160.000, Y  +517.221, Z    +0.000, E1   -21.778, E3 +13369.581}
SPL {X  -160.000, Y  +521.677, Z    +0.000, E1   -21.781, E3 +13393.342}
SPL {X  -160.000, Y  +525.729, Z    +0.000, E1   -21.753, E3 +13414.981}
SPL {X  -160.000, Y  +529.456, Z    +0.000, E1   -21.766, E3 +13434.761}
SPL {X  -160.000, Y  +533.608, Z    +0.000, E1   -21.776, E3 +13456.891}
SPL {X  -160.000, Y  +538.227, Z    +0.000, E1   -21.794, E3 +13481.423}
SPL {X  -160.000, Y  +542.483, Z    +0.000, E1   -21.764, E3 +13504.149}
SPL {X  -160.000, Y  +546.194, Z    +0.000, E1   -21.754, E3 +13523.965}
SPL {X  -160.000, Y  +550.131, Z    +0.000, E1   -21.771, E3 +13544.901}
SPL {X  -160.000, Y  +554.462, Z    +0.000, E1   -21.777, E3 +13567.955}
SPL {X  -160.000, Y  +558.542, Z    +0.000, E1   -21.758, E3 +13589.727}
SPL {X  -160.000, Y  +562.615, Z    +0.000, E1   -21.776, E3 +13611.383}
SPL {X  -160.000, Y  +566.764, Z    +0.000, E1   -21.764, E3 +13633.508}
SPL {X  -160.000, Y  +570.657, Z    +0.000, E1   -21.758, E3 +13654.256}
SPL {X  -160.000, Y  +574.688, Z    +0.000, E1   -21.771, E3 +13675.698}
SPL {X  -160.000, Y  +578.864, Z    +0.000, E1   -21.770, E3 +13697.949}
SPL {X  -160.000, Y  +582.807, Z    +0.000, E1   -21.754, E3 +13719.003}
SPL {X  -160.000, Y  +586.993, Z    +0.000, E1   -21.779, E3 +13741.239}
SPL {X  -160.000, Y  +591.368, Z    +0.000, E1   -21.775, E3 +13764.526}
SPL {X  -160.000, Y  +595.703, Z    +0.000, E1   -21.775, E3 +13787.635}
SPL {X  -160.000, Y  +599.558, Z    +0.000, E1   -21.748, E3 +13808.213}
SPL {X  -160.000, Y  +603.126, Z    +0.000, E1   -21.757, E3 +13827.192}
SPL {X  -160.000, Y  +607.107, Z    +0.000, E1   -21.766, E3 +13848.418}
SPL {X  -160.000, Y  +611.246, Z    +0.000, E1   -21.760, E3 +13870.491}
SPL {X  -160.000, Y  +615.151, Z    +0.000, E1   -21.752, E3 +13891.304}
SPL {X  -160.000, Y  +618.728, Z    +0.000, E1   -21.747, E3 +13910.367}
SPL {X  -160.000, Y  +622.318, Z    +0.000, E1   -21.753, E3 +13929.481}
SPL {X  -160.000, Y  +625.877, Z    +0.000, E1   -21.745, E3 +13948.459}
SPL {X  -160.000, Y  +629.892, Z    +0.000, E1   -21.777, E3 +13969.783}
SPL {X  -160.000, Y  +634.024, Z    +0.000, E1   -21.756, E3 +13991.834}
SPL {X  -160.000, Y  +637.661, Z    +0.000, E1   -21.748, E3 +14011.224}
SPL {X  -160.000, Y  +641.244, Z    +0.000, E1   -21.752, E3 +14030.295}
SPL {X  -160.000, Y  +645.120, Z    +0.000, E1   -21.762, E3 +14050.927}
SPL {X  -160.000, Y  +649.214, Z    +0.000, E1   -21.766, E3 +14072.715}
SPL {X  -160.000, Y  +653.188, Z    +0.000, E1   -21.771, E3 +14093.778}
SPL {X  -160.000, Y  +656.905, Z    +0.000, E1   -21.769, E3 +14113.553}
SPL {X  -160.000, Y  +660.685, Z    +0.000, E1   -21.769, E3 +14133.721}
SPL {X  -160.000, Y  +664.985, Z    +0.000, E1   -21.790, E3 +14156.574}
SPL {X  -159.993, Y  +669.170, Z    +0.000, E1   -21.763, E3 +14178.933}
SPL {X  -159.916, Y  +672.869, Z    +0.000, E1   -21.755, E3 +14198.677}
SPL {X  -159.752, Y  +676.610, Z    +0.000, E1   -21.740, E3 +14218.752}
SPL {X  -159.478, Y  +680.618, Z    +0.000, E1   -21.719, E3 +14240.351}
SPL {X  -159.108, Y  +684.576, Z    +0.000, E1   -21.664, E3 +14261.821}
SPL {X  -158.638, Y  +688.530, Z    +0.000, E1   -21.617, E3 +14283.342}
SPL {X  -158.097, Y  +692.303, Z    +0.000, E1   -21.529, E3 +14304.060}
ENDSPLINE

SPLINE
SPL {X  -158.264, Y  +691.203, Z    +0.000, E1   -17.264, E3 +14340.805}
SPL {X  -159.000, Y  +685.560, Z    +0.000, E1   -12.398, E3 +14361.981}
SPL {X  -159.924, Y  +672.625, Z    +0.000, E1    -3.689, E3 +14376.998}
SPL {X  -160.000, Y  +663.203, Z    +0.000, E1    +3.155, E3 +14383.652}
SPL {X  -160.000, Y  +652.103, Z    +0.000, E1   +11.247, E3 +14395.322}
SPL {X  -160.000, Y  +641.822, Z    +0.000, E1   +17.059, E3 +14414.696}
SPL {X  -160.000, Y  +631.293, Z    +0.000, E1   +20.354, E3 +14448.576}
SPL {X  -160.000, Y  +627.542, Z    +0.000, E1   +20.380, E3 +14469.983}
SPL {X  -160.000, Y  +623.532, Z    +0.000, E1   +20.378, E3 +14492.948}
SPL {X  -160.000, Y  +619.329, Z    +0.000, E1   +20.391, E3 +14516.986}
SPL {X  -160.000, Y  +614.967, Z    +0.000, E1   +20.392, E3 +14541.966}
SPL {X  -160.000, Y  +611.206, Z    +0.000, E1   +20.351, E3 +14563.638}
SPL {X  -160.000, Y  +607.824, Z    +0.000, E1   +20.354, E3 +14583.058}
SPL {X  -160.000, Y  +603.899, Z    +0.000, E1   +20.373, E3 +14605.508}
SPL {X  -160.000, Y  +599.617, Z    +0.000, E1   +20.384, E3 +14630.002}
SPL {X  -160.000, Y  +595.532, Z    +0.000, E1   +20.373, E3 +14653.363}
SPL {X  -160.000, Y  +591.705, Z    +0.000, E1   +20.373, E3 +14675.287}
SPL {X  -160.000, Y  +588.037, Z    +0.000, E1   +20.359, E3 +14696.374}
SPL {X  -160.000, Y  +584.320, Z    +0.000, E1   +20.364, E3 +14717.676}
SPL {X  -160.000, Y  +580.616, Z    +0.000, E1   +20.357, E3 +14738.903}
SPL {X  -160.000, Y  +577.083, Z    +0.000, E1   +20.358, E3 +14759.151}
SPL {X  -160.000, Y  +573.158, Z    +0.000, E1   +20.377, E3 +14781.604}
SPL {X  -160.000, Y  +568.802, Z    +0.000, E1   +20.385, E3 +14806.555}
SPL {X  -160.000, Y  +564.937, Z    +0.000, E1   +20.350, E3 +14828.776}
SPL {X  -160.000, Y  +561.213, Z    +0.000, E1   +20.372, E3 +14850.062}
SPL {X  -160.000, Y  +557.320, Z    +0.000, E1   +20.363, E3 +14872.389}
SPL {X  -160.000, Y  +553.712, Z    +0.000, E1   +20.355, E3 +14893.088}
SPL {X  -160.000, Y  +550.040, Z    +0.000, E1   +20.360, E3 +14914.127}
SPL {X  -160.000, Y  +546.180, Z    +0.000, E1   +20.370, E3 +14936.182}
SPL {X  -160.000, Y  +542.032, Z    +0.000, E1   +20.384, E3 +14959.921}
SPL {X  -160.000, Y  +537.870, Z    +0.000, E1   +20.372, E3 +14983.797}
SPL {X  -160.000, Y  +534.086, Z    +0.000, E1   +20.356, E3 +15005.551}
SPL {X  -160.000, Y  +530.164, Z    +0.000, E1   +20.382, E3 +15027.900}
SPL {X  -160.000, Y  +527.505, Z    +0.000, E1   +20.318, E3 +15043.274}
SPL {X  -160.000, Y  +511.620, Z    +0.000, E1   +28.365, E3 +15053.737}
SPL {X  -160.000, Y  +507.906, Z    +0.000, E1   +28.152, E3 +15070.132}
SPL {X  -160.000, Y  +506.085, Z    +0.000, E1   +26.146, E3 +15092.592}
SPL {X  -160.000, Y  +504.342, Z    +0.000, E1   +24.109, E3 +15116.107}
SPL {X  -160.000, Y  +503.002, Z    +0.000, E1   +22.325, E3 +15137.112}
SPL {X  -160.000, Y  +500.783, Z    +0.000, E1   +21.421, E3 +15156.702}
SPL {X  -160.000, Y  +497.229, Z    +0.000, E1   +21.403, E3 +15176.010}
SPL {X  -160.000, Y  +493.901, Z    +0.000, E1   +21.409, E3 +15194.029}
SPL {X  -160.000, Y  +490.791, Z    +0.000, E1   +21.400, E3 +15210.902}
SPL {X  -160.000, Y  +487.647, Z    +0.000, E1   +21.401, E3 +15227.948}
SPL {X  -160.000, Y  +484.273, Z    +0.000, E1   +21.408, E3 +15246.228}
SPL {X  -160.000, Y  +481.093, Z    +0.000, E1   +21.389, E3 +15263.537}
SPL {X  -160.000, Y  +478.021, Z    +0.000, E1   +21.401, E3 +15280.143}
SPL {X  -160.000, Y  +474.639, Z    +0.000, E1   +21.410, E3 +15298.435}
SPL {X  -160.000, Y  +471.343, Z    +0.000, E1   +21.399, E3 +15316.337}
SPL {X  -160.000, Y  +468.133, Z    +0.000, E1   +21.402, E3 +15333.728}
SPL {X  -160.000, Y  +464.638, Z    +0.000, E1   +21.421, E3 +15352.578}
SPL {X  -160.000, Y  +461.045, Z    +0.000, E1   +21.424, E3 +15371.991}
SPL {X  -160.000, Y  +457.606, Z    +0.000, E1   +21.413, E3 +15390.701}
SPL {X  -160.000, Y  +454.417, Z    +0.000, E1   +21.401, E3 +15408.010}
SPL {X  -160.000, Y  +451.425, Z    +0.000, E1   +21.404, E3 +15424.231}
SPL {X  -160.000, Y  +448.039, Z    +0.000, E1   +21.417, E3 +15442.524}
SPL {X  -160.000, Y  +444.787, Z    +0.000, E1   +21.414, E3 +15460.080}
SPL {X  -160.000, Y  +441.637, Z    +0.000, E1   +21.431, E3 +15477.058}
SPL {X  -160.000, Y  +438.199, Z    +0.000, E1   +21.432, E3 +15495.662}
SPL {X  -160.000, Y  +434.875, Z    +0.000, E1   +21.424, E3 +15513.701}
SPL {X  -160.000, Y  +431.689, Z    +0.000, E1   +21.423, E3 +15530.950}
SPL {X  -160.000, Y  +428.451, Z    +0.000, E1   +21.430, E3 +15548.429}
SPL {X  -160.000, Y  +425.120, Z    +0.000, E1   +21.430, E3 +15566.494}
SPL {X  -160.000, Y  +421.671, Z    +0.000, E1   +21.430, E3 +15585.178}
SPL {X  -160.000, Y  +418.225, Z    +0.000, E1   +21.425, E3 +15603.859}
SPL {X  -160.000, Y  +414.956, Z    +0.000, E1   +21.424, E3 +15621.540}
SPL {X  -160.000, Y  +411.834, Z    +0.000, E1   +21.420, E3 +15638.458}
SPL {X  -160.000, Y  +408.570, Z    +0.000, E1   +21.432, E3 +15656.067}
SPL {X  -160.000, Y  +405.237, Z    +0.000, E1   +21.432, E3 +15674.096}
SPL {X  -160.000, Y  +402.004, Z    +0.000, E1   +21.424, E3 +15691.671}
SPL {X  -160.000, Y  +398.626, Z    +0.000, E1   +21.425, E3 +15709.977}
SPL {X  -160.000, Y  +395.405, Z    +0.000, E1   +21.422, E3 +15727.394}
SPL {X  -160.000, Y  +392.641, Z    +0.000, E1   +21.407, E3 +15742.393}
SPL {X  -159.989, Y  +390.129, Z    +0.000, E1   +21.406, E3 +15756.034}
SPL {X  -159.932, Y  +387.337, Z    +0.000, E1   +21.403, E3 +15771.229}
SPL {X  -159.823, Y  +384.478, Z    +0.000, E1   +21.379, E3 +15786.893}
SPL {X  -159.660, Y  +381.581, Z    +0.000, E1   +21.363, E3 +15802.781}
SPL {X  -159.452, Y  +378.773, Z    +0.000, E1   +21.330, E3 +15818.228}
SPL {X  -159.222, Y  +376.244, Z    +0.000, E1   +21.297, E3 +15832.190}
SPL {X  -158.814, Y  +372.556, Z    +0.000, E1   +21.316, E3 +15852.457}
SPL {X  -158.301, Y  +368.743, Z    +0.000, E1   +21.199, E3 +15873.779}
SPL {X  -157.981, Y  +366.660, Z    +0.000, E1   +19.986, E3 +15896.746}
ENDSPLINE

SPLINE
SPL {X  -158.491, Y  +370.077, Z    +0.000, E1   +15.910, E3 +15921.759}
SPL {X  -159.771, Y  +383.450, Z    +0.000, E1    +6.314, E3 +15944.915}
SPL {X  -160.000, Y  +392.463, Z    +0.000, E1    +0.112, E3 +15951.422}
SPL {X  -160.000, Y  +399.874, Z    +0.000, E1    -5.508, E3 +15955.924}
SPL {X  -160.000, Y  +411.622, Z    +0.000, E1   -13.815, E3 +15968.044}
SPL {X  -160.000, Y  +419.836, Z    +0.000, E1   -18.198, E3 +15983.218}
SPL {X  -160.000, Y  +430.523, Z    +0.000, E1   -21.710, E3 +16013.418}
SPL {X  -160.000, Y  +433.426, Z    +0.000, E1   -21.735, E3 +16028.832}
SPL {X  -160.000, Y  +436.131, Z    +0.000, E1   -21.710, E3 +16043.307}
SPL {X  -160.000, Y  +439.046, Z    +0.000, E1   -21.732, E3 +16058.800}
SPL {X  -160.000, Y  +442.009, Z    +0.000, E1   -21.719, E3 +16074.622}
SPL {X  -160.000, Y  +444.891, Z    +0.000, E1   -21.724, E3 +16089.978}
SPL {X  -160.000, Y  +449.017, Z    +0.000, E1   -21.792, E3 +16111.770}
SPL {X  -160.000, Y  +452.864, Z    +0.000, E1   -21.730, E3 +16132.387}
SPL {X  -160.000, Y  +455.470, Z    +0.000, E1   -21.722, E3 +16146.276}
SPL {X  -160.000, Y  +458.295, Z    +0.000, E1   -21.738, E3 +16161.297}
SPL {X  -160.000, Y  +461.133, Z    +0.000, E1   -21.720, E3 +16176.480}
SPL {X  -160.000, Y  +464.458, Z    +0.000, E1   -21.770, E3 +16193.999}
SPL {X  -160.000, Y  +468.250, Z    +0.000, E1   -21.764, E3 +16214.152}
SPL {X  -160.000, Y  +472.226, Z    +0.000, E1   -21.782, E3 +16235.310}
SPL {X  -160.000, Y  +476.333, Z    +0.000, E1   -21.767, E3 +16257.225}
SPL {X  -160.000, Y  +480.244, Z    +0.000, E1   -21.765, E3 +16278.089}
SPL {X  -160.000, Y  +484.301, Z    +0.000, E1   -21.775, E3 +16299.618}
SPL {X  -160.000, Y  +488.201, Z    +0.000, E1   -21.768, E3 +16320.378}
SPL {X  -160.000, Y  +492.394, Z    +0.000, E1   -21.802, E3 +16342.552}
SPL {X  -160.000, Y  +496.781, Z    +0.000, E1   -21.798, E3 +16365.863}
SPL {X  -160.000, Y  +501.083, Z    +0.000, E1   -21.796, E3 +16388.793}
SPL {X  -160.000, Y  +504.917, Z    +0.000, E1   -21.764, E3 +16409.298}
SPL {X  -160.000, Y  +508.886, Z    +0.000, E1   -21.791, E3 +16430.384}
SPL {X  -160.000, Y  +513.057, Z    +0.000, E1   -21.767, E3 +16452.691}
SPL {X  -160.000, Y  +517.221, Z    +0.000, E1   -21.778, E3 +16474.844}
SPL {X  -160.000, Y  +521.677, Z    +0.000, E1   -21.781, E3 +16498.605}
SPL {X  -160.000, Y  +525.729, Z    +0.000, E1   -21.753, E3 +16520.245}
SPL {X  -160.000, Y  +529.456, Z    +0.000, E1   -21.766, E3 +16540.024}
SPL {X  -160.000, Y  +533.608, Z    +0.000, E1   -21.776, E3 +16562.154}
SPL {X  -160.000, Y  +538.227, Z    +0.000, E1   -21.794, E3 +16586.687}
SPL {X  -160.000, Y  +542.483, Z    +0.000, E1   -21.764, E3 +16609.412}
SPL {X  -160.000, Y  +546.194, Z    +0.000, E1   -21.754, E3 +16629.229}
SPL {X  -160.000, Y  +550.131, Z    +0.000, E1   -21.771, E3 +16650.164}
SPL {X  -160.000, Y  +554.462, Z    +0.000, E1   -21.777, E3 +16673.218}
SPL {X  -160.000, Y  +558.542, Z    +0.000, E1   -21.758, E3 +16694.991}
SPL {X  -160.000, Y  +562.615, Z    +0.000, E1   -21.776, E3 +16716.647}
SPL {X  -160.000, Y  +566.764, Z    +0.000, E1   -21.764, E3 +16738.772}
SPL {X  -160.000, Y  +570.657, Z    +0.000, E1   -21.758, E3 +16759.519}
SPL {X  -160.000, Y  +574.688, Z    +0.000, E1   -21.771, E3 +16780.962}
SPL {X  -160.000, Y  +578.864, Z    +0.000, E1   -21.770, E3 +16803.213}
SPL {X  -160.000, Y  +582.807, Z    +0.000, E1   -21.754, E3 +16824.267}
SPL {X  -160.000, Y  +586.993, Z    +0.000, E1   -21.779, E3 +16846.502}
SPL {X  -160.000, Y  +591.368, Z    +0.000, E1   -21.775, E3 +16869.789}
SPL {X  -160.000, Y  +595.703, Z    +0.000, E1   -21.775, E3 +16892.899}
SPL {X  -160.000, Y  +599.558, Z    +0.000, E1   -21.748, E3 +16913.476}
SPL {X  -160.000, Y  +603.126, Z    +0.000, E1   -21.757, E3 +16932.456}
SPL {X  -160.000, Y  +607.107, Z    +0.000, E1   -21.766, E3 +16953.681}
SPL {X  -160.000, Y  +611.246, Z    +0.000, E1   -21.760, E3 +16975.754}
SPL {X  -160.000, Y  +615.151, Z    +0.000, E1   -21.752, E3 +16996.568}
SPL {X  -160.000, Y  +618.728, Z    +0.000, E1   -21.747, E3 +17015.630}
SPL {X  -160.000, Y  +622.318, Z    +0.000, E1   -21.753, E3 +17034.745}
SPL {X  -160.000, Y  +625.877, Z    +0.000, E1   -21.745, E3 +17053.723}
SPL {X  -160.000, Y  +629.892, Z    +0.000, E1   -21.777, E3 +17075.047}
SPL {X  -160.000, Y  +634.024, Z    +0.000, E1   -21.756, E3 +17097.097}
SPL {X  -160.000, Y  +637.661, Z    +0.000, E1   -21.748, E3 +17116.488}
SPL {X  -160.000, Y  +641.244, Z    +0.000, E1   -21.752, E3 +17135.558}
SPL {X  -160.000, Y  +645.120, Z    +0.000, E1   -21.762, E3 +17156.191}
SPL {X  -160.000, Y  +649.214, Z    +0.000, E1   -21.766, E3 +17177.979}
SPL {X  -160.000, Y  +653.188, Z    +0.000, E1   -21.771, E3 +17199.041}
SPL {X  -160.000, Y  +656.905, Z    +0.000, E1   -21.769, E3 +17218.817}
SPL {X  -160.000, Y  +660.685, Z    +0.000, E1   -21.769, E3 +17238.985}
SPL {X  -160.000, Y  +664.985, Z    +0.000, E1   -21.790, E3 +17261.837}
SPL {X  -159.993, Y  +669.170, Z    +0.000, E1   -21.763, E3 +17284.196}
SPL {X  -159.916, Y  +672.869, Z    +0.000, E1   -21.755, E3 +17303.941}
SPL {X  -159.752, Y  +676.610, Z    +0.000, E1   -21.740, E3 +17324.016}
SPL {X  -159.478, Y  +680.618, Z    +0.000, E1   -21.719, E3 +17345.615}
SPL {X  -159.108, Y  +684.576, Z    +0.000, E1   -21.664, E3 +17367.084}
SPL {X  -158.638, Y  +688.530, Z    +0.000, E1   -21.617, E3 +17388.606}
SPL {X  -158.097, Y  +692.303, Z    +0.000, E1   -21.529, E3 +17409.324}
ENDSPLINE

SPLINE
SPL {X  -158.264, Y  +691.203, Z    +0.000, E1   -17.264, E3 +17446.069}
SPL {X  -159.000, Y  +685.560, Z    +0.000, E1   -12.398, E3 +17467.244}
SPL {X  -159.924, Y  +672.625, Z    +0.000, E1    -3.689, E3 +17482.261}
SPL {X  -160.000, Y  +663.203, Z    +0.000, E1    +3.155, E3 +17488.916}
SPL {X  -160.000, Y  +652.103, Z    +0.000, E1   +11.247, E3 +17500.586}
SPL {X  -160.000, Y  +641.822, Z    +0.000, E1   +17.059, E3 +17519.960}
SPL {X  -160.000, Y  +631.293, Z    +0.000, E1   +20.354, E3 +17553.839}
SPL {X  -160.000, Y  +627.542, Z    +0.000, E1   +20.380, E3 +17575.246}
SPL {X  -160.000, Y  +623.532, Z    +0.000, E1   +20.378, E3 +17598.212}
SPL {X  -160.000, Y  +619.329, Z    +0.000, E1   +20.391, E3 +17622.250}
SPL {X  -160.000, Y  +614.967, Z    +0.000, E1   +20.392, E3 +17647.229}
SPL {X  -160.000, Y  +611.206, Z    +0.000, E1   +20.351, E3 +17668.901}
SPL {X  -160.000, Y  +607.824, Z    +0.000, E1   +20.354, E3 +17688.322}
SPL {X  -160.000, Y  +603.899, Z    +0.000, E1   +20.373, E3 +17710.772}
SPL {X  -160.000, Y  +599.617, Z    +0.000, E1   +20.384, E3 +17735.266}
SPL {X  -160.000, Y  +595.532, Z    +0.000, E1   +20.373, E3 +17758.626}
SPL {X  -160.000, Y  +591.705, Z    +0.000, E1   +20.373, E3 +17780.551}
SPL {X  -160.000, Y  +588.037, Z    +0.000, E1   +20.359, E3 +17801.638}
SPL {X  -160.000, Y  +584.320, Z    +0.000, E1   +20.364, E3 +17822.939}
SPL {X  -160.000, Y  +580.616, Z    +0.000, E1   +20.357, E3 +17844.166}
SPL {X  -160.000, Y  +577.083, Z    +0.000, E1   +20.358, E3 +17864.415}
SPL {X  -160.000, Y  +573.158, Z    +0.000, E1   +20.377, E3 +17886.867}
SPL {X  -160.000, Y  +568.802, Z    +0.000, E1   +20.385, E3 +17911.819}
SPL {X  -160.000, Y  +564.937, Z    +0.000, E1   +20.350, E3 +17934.039}
SPL {X  -160.000, Y  +561.213, Z    +0.000, E1   +20.372, E3 +17955.326}
SPL {X  -160.000, Y  +557.320, Z    +0.000, E1   +20.363, E3 +17977.653}
SPL {X  -160.000, Y  +553.712, Z    +0.000, E1   +20.355, E3 +17998.352}
SPL {X  -160.000, Y  +550.040, Z    +0.000, E1   +20.360, E3 +18019.390}
SPL {X  -160.000, Y  +546.180, Z    +0.000, E1   +20.370, E3 +18041.446}
SPL {X  -160.000, Y  +542.032, Z    +0.000, E1   +20.384, E3 +18065.185}
SPL {X  -160.000, Y  +537.870, Z    +0.000, E1   +20.372, E3 +18089.060}
SPL {X  -160.000, Y  +534.086, Z    +0.000, E1   +20.356, E3 +18110.814}
SPL {X  -160.000, Y  +530.164, Z    +0.000, E1   +20.382, E3 +18133.164}
SPL {X  -160.000, Y  +527.505, Z    +0.000, E1   +20.318, E3 +18148.538}
SPL {X  -160.000, Y  +511.620, Z    +0.000, E1   +28.365, E3 +18159.001}
SPL {X  -160.000, Y  +507.906, Z    +0.000, E1   +28.152, E3 +18175.396}
SPL {X  -160.000, Y  +506.085, Z    +0.000, E1   +26.146, E3 +18197.855}
SPL {X  -160.000, Y  +504.342, Z    +0.000, E1   +24.109, E3 +18221.370}
SPL {X  -160.000, Y  +503.002, Z    +0.000, E1   +22.325, E3 +18242.376}
SPL {X  -160.000, Y  +500.783, Z    +0.000, E1   +21.421, E3 +18261.965}
SPL {X  -160.000, Y  +497.229, Z    +0.000, E1   +21.403, E3 +18281.273}
SPL {X  -160.000, Y  +493.901, Z    +0.000, E1   +21.409, E3 +18299.292}
SPL {X  -160.000, Y  +490.791, Z    +0.000, E1   +21.400, E3 +18316.165}
SPL {X  -160.000, Y  +487.647, Z    +0.000, E1   +21.401, E3 +18333.211}
SPL {X  -160.000, Y  +484.273, Z    +0.000, E1   +21.408, E3 +18351.491}
SPL {X  -160.000, Y  +481.093, Z    +0.000, E1   +21.389, E3 +18368.800}
SPL {X  -160.000, Y  +478.021, Z    +0.000, E1   +21.401, E3 +18385.407}
SPL {X  -160.000, Y  +474.639, Z    +0.000, E1   +21.410, E3 +18403.698}
SPL {X  -160.000, Y  +471.343, Z    +0.000, E1   +21.399, E3 +18421.600}
SPL {X  -160.000, Y  +468.133, Z    +0.000, E1   +21.402, E3 +18438.992}
SPL {X  -160.000, Y  +464.638, Z    +0.000, E1   +21.421, E3 +18457.841}
SPL {X  -160.000, Y  +461.045, Z    +0.000, E1   +21.424, E3 +18477.255}
SPL {X  -160.000, Y  +457.606, Z    +0.000, E1   +21.413, E3 +18495.965}
SPL {X  -160.000, Y  +454.417, Z    +0.000, E1   +21.401, E3 +18513.273}
SPL {X  -160.000, Y  +451.425, Z    +0.000, E1   +21.404, E3 +18529.495}
SPL {X  -160.000, Y  +448.039, Z    +0.000, E1   +21.417, E3 +18547.788}
SPL {X  -160.000, Y  +444.787, Z    +0.000, E1   +21.414, E3 +18565.343}
SPL {X  -160.000, Y  +441.637, Z    +0.000, E1   +21.431, E3 +18582.321}
SPL {X  -160.000, Y  +438.199, Z    +0.000, E1   +21.432, E3 +18600.925}
SPL {X  -160.000, Y  +434.875, Z    +0.000, E1   +21.424, E3 +18618.965}
SPL {X  -160.000, Y  +431.689, Z    +0.000, E1   +21.423, E3 +18636.213}
SPL {X  -160.000, Y  +428.451, Z    +0.000, E1   +21.430, E3 +18653.693}
SPL {X  -160.000, Y  +425.120, Z    +0.000, E1   +21.430, E3 +18671.757}
SPL {X  -160.000, Y  +421.671, Z    +0.000, E1   +21.430, E3 +18690.441}
SPL {X  -160.000, Y  +418.225, Z    +0.000, E1   +21.425, E3 +18709.123}
SPL {X  -160.000, Y  +414.956, Z    +0.000, E1   +21.424, E3 +18726.803}
SPL {X  -160.000, Y  +411.834, Z    +0.000, E1   +21.420, E3 +18743.722}
SPL {X  -160.000, Y  +408.570, Z    +0.000, E1   +21.432, E3 +18761.331}
SPL {X  -160.000, Y  +405.237, Z    +0.000, E1   +21.432, E3 +18779.359}
SPL {X  -160.000, Y  +402.004, Z    +0.000, E1   +21.424, E3 +18796.934}
SPL {X  -160.000, Y  +398.626, Z    +0.000, E1   +21.425, E3 +18815.241}
SPL {X  -160.000, Y  +395.405, Z    +0.000, E1   +21.422, E3 +18832.658}
SPL {X  -160.000, Y  +392.641, Z    +0.000, E1   +21.407, E3 +18847.656}
SPL {X  -159.989, Y  +390.129, Z    +0.000, E1   +21.406, E3 +18861.297}
SPL {X  -159.932, Y  +387.337, Z    +0.000, E1   +21.403, E3 +18876.493}
SPL {X  -159.823, Y  +384.478, Z    +0.000, E1   +21.379, E3 +18892.156}
SPL {X  -159.660, Y  +381.581, Z    +0.000, E1   +21.363, E3 +18908.044}
SPL {X  -159.452, Y  +378.773, Z    +0.000, E1   +21.330, E3 +18923.491}
SPL {X  -159.222, Y  +376.244, Z    +0.000, E1   +21.297, E3 +18937.453}
SPL {X  -158.814, Y  +372.556, Z    +0.000, E1   +21.316, E3 +18957.720}
SPL {X  -158.301, Y  +368.743, Z    +0.000, E1   +21.199, E3 +18979.042}
SPL {X  -157.981, Y  +366.660, Z    +0.000, E1   +19.986, E3 +19002.010}
ENDSPLINE

SPLINE
SPL {X  -158.491, Y  +370.077, Z    +0.000, E1   +15.910, E3 +19027.023}
SPL {X  -159.771, Y  +383.450, Z    +0.000, E1    +6.314, E3 +19050.178}
SPL {X  -160.000, Y  +392.463, Z    +0.000, E1    +0.112, E3 +19056.685}
SPL {X  -160.000, Y  +399.874, Z    +0.000, E1    -5.508, E3 +19061.187}
SPL {X  -160.000, Y  +411.622, Z    +0.000, E1   -13.815, E3 +19073.307}
SPL {X  -160.000, Y  +419.836, Z    +0.000, E1   -18.198, E3 +19088.481}
SPL {X  -160.000, Y  +430.523, Z    +0.000, E1   -21.710, E3 +19118.681}
SPL {X  -160.000, Y  +433.426, Z    +0.000, E1   -21.735, E3 +19134.096}
SPL {X  -160.000, Y  +436.131, Z    +0.000, E1   -21.710, E3 +19148.571}
SPL {X  -160.000, Y  +439.046, Z    +0.000, E1   -21.732, E3 +19164.064}
SPL {X  -160.000, Y  +442.009, Z    +0.000, E1   -21.719, E3 +19179.886}
SPL {X  -160.000, Y  +444.891, Z    +0.000, E1   -21.724, E3 +19195.242}
SPL {X  -160.000, Y  +449.017, Z    +0.000, E1   -21.792, E3 +19217.033}
SPL {X  -160.000, Y  +452.864, Z    +0.000, E1   -21.730, E3 +19237.651}
SPL {X  -160.000, Y  +455.470, Z    +0.000, E1   -21.722, E3 +19251.540}
SPL {X  -160.000, Y  +458.295, Z    +0.000, E1   -21.738, E3 +19266.561}
SPL {X  -160.000, Y  +461.133, Z    +0.000, E1   -21.720, E3 +19281.744}
SPL {X  -160.000, Y  +464.458, Z    +0.000, E1   -21.770, E3 +19299.262}
SPL {X  -160.000, Y  +468.250, Z    +0.000, E1   -21.764, E3 +19319.416}
SPL {X  -160.000, Y  +472.226, Z    +0.000, E1   -21.782, E3 +19340.574}
SPL {X  -160.000, Y  +476.333, Z    +0.000, E1   -21.767, E3 +19362.488}
SPL {X  -160.000, Y  +480.244, Z    +0.000, E1   -21.765, E3 +19383.353}
SPL {X  -160.000, Y  +484.301, Z    +0.000, E1   -21.775, E3 +19404.881}
SPL {X  -160.000, Y  +488.201, Z    +0.000, E1   -21.768, E3 +19425.641}
SPL {X  -160.000, Y  +492.394, Z    +0.000, E1   -21.802, E3 +19447.816}
SPL {X  -160.000, Y  +496.781, Z    +0.000, E1   -21.798, E3 +19471.127}
SPL {X  -160.000, Y  +501.083, Z    +0.000, E1   -21.796, E3 +19494.057}
SPL {X  -160.000, Y  +504.917, Z    +0.000, E1   -21.764, E3 +19514.561}
SPL {X  -160.000, Y  +508.886, Z    +0.000, E1   -21.791, E3 +19535.647}
SPL {X  -160.000, Y  +513.057, Z    +0.000, E1   -21.767, E3 +19557.955}
SPL {X  -160.000, Y  +517.221, Z    +0.000, E1   -21.778, E3 +19580.108}
SPL {X  -160.000, Y  +521.677, Z    +0.000, E1   -21.781, E3 +19603.869}
SPL {X  -160.000, Y  +525.729, Z    +0.000, E1   -21.753, E3 +19625.508}
SPL {X  -160.000, Y  +529.456, Z    +0.000, E1   -21.766, E3 +19645.288}
SPL {X  -160.000, Y  +533.608, Z    +0.000, E1   -21.776, E3 +19667.418}
SPL {X  -160.000, Y  +538.227, Z    +0.000, E1   -21.794, E3 +19691.950}
SPL {X  -160.000, Y  +542.483, Z    +0.000, E1   -21.764, E3 +19714.676}
SPL {X  -160.000, Y  +546.194, Z    +0.000, E1   -21.754, E3 +19734.492}
SPL {X  -160.000, Y  +550.131, Z    +0.000, E1   -21.771, E3 +19755.428}
SPL {X  -160.000, Y  +554.462, Z    +0.000, E1   -21.777, E3 +19778.482}
SPL {X  -160.000, Y  +558.542, Z    +0.000, E1   -21.758, E3 +19800.254}
SPL {X  -160.000, Y  +562.615, Z    +0.000, E1   -21.776, E3 +19821.910}
SPL {X  -160.000, Y  +566.764, Z    +0.000, E1   -21.764, E3 +19844.035}
SPL {X  -160.000, Y  +570.657, Z    +0.000, E1   -21.758, E3 +19864.783}
SPL {X  -160.000, Y  +574.688, Z    +0.000, E1   -21.771, E3 +19886.225}
SPL {X  -160.000, Y  +578.864, Z    +0.000, E1   -21.770, E3 +19908.476}
SPL {X  -160.000, Y  +582.807, Z    +0.000, E1   -21.754, E3 +19929.530}
SPL {X  -160.000, Y  +586.993, Z    +0.000, E1   -21.779, E3 +19951.766}
SPL {X  -160.000, Y  +591.368, Z    +0.000, E1   -21.775, E3 +19975.053}
SPL {X  -160.000, Y  +595.703, Z    +0.000, E1   -21.775, E3 +19998.163}
SPL {X  -160.000, Y  +599.558, Z    +0.000, E1   -21.748, E3 +20018.740}
SPL {X  -160.000, Y  +603.126, Z    +0.000, E1   -21.757, E3 +20037.719}
SPL {X  -160.000, Y  +607.107, Z    +0.000, E1   -21.766, E3 +20058.945}
SPL {X  -160.000, Y  +611.246, Z    +0.000, E1   -21.760, E3 +20081.018}
SPL {X  -160.000, Y  +615.151, Z    +0.000, E1   -21.752, E3 +20101.831}
SPL {X  -160.000, Y  +618.728, Z    +0.000, E1   -21.747, E3 +20120.894}
SPL {X  -160.000, Y  +622.318, Z    +0.000, E1   -21.753, E3 +20140.008}
SPL {X  -160.000, Y  +625.877, Z    +0.000, E1   -21.745, E3 +20158.987}
SPL {X  -160.000, Y  +629.892, Z    +0.000, E1   -21.777, E3 +20180.310}
SPL {X  -160.000, Y  +634.024, Z    +0.000, E1   -21.756, E3 +20202.361}
SPL {X  -160.000, Y  +637.661, Z    +0.000, E1   -21.748, E3 +20221.751}
SPL {X  -160.000, Y  +641.244, Z    +0.000, E1   -21.752, E3 +20240.822}
SPL {X  -160.000, Y  +645.120, Z    +0.000, E1   -21.762, E3 +20261.454}
SPL {X  -160.000, Y  +649.214, Z    +0.000, E1   -21.766, E3 +20283.243}
SPL {X  -160.000, Y  +653.188, Z    +0.000, E1   -21.771, E3 +20304.305}
SPL {X  -160.000, Y  +656.905, Z    +0.000, E1   -21.769, E3 +20324.080}
SPL {X  -160.000, Y  +660.685, Z    +0.000, E1   -21.769, E3 +20344.248}
SPL {X  -160.000, Y  +664.985, Z    +0.000, E1   -21.790, E3 +20367.101}
SPL {X  -159.993, Y  +669.170, Z    +0.000, E1   -21.763, E3 +20389.460}
SPL {X  -159.916, Y  +672.869, Z    +0.000, E1   -21.755, E3 +20409.204}
SPL {X  -159.752, Y  +676.610, Z    +0.000, E1   -21.740, E3 +20429.279}
SPL {X  -159.478, Y  +680.618, Z    +0.000, E1   -21.719, E3 +20450.879}
SPL {X  -159.108, Y  +684.576, Z    +0.000, E1   -21.664, E3 +20472.348}
SPL {X  -158.638, Y  +688.530, Z    +0.000, E1   -21.617, E3 +20493.869}
SPL {X  -158.097, Y  +692.303, Z    +0.000, E1   -21.529, E3 +20514.587}
ENDSPLINE

SPLINE
SPL {X  -158.264, Y  +691.203, Z    +0.000, E1   -17.264, E3 +20551.332}
SPL {X  -159.000, Y  +685.560, Z    +0.000, E1   -12.398, E3 +20572.508}
SPL {X  -159.924, Y  +672.625, Z    +0.000, E1    -3.689, E3 +20587.525}
SPL {X  -160.000, Y  +663.203, Z    +0.000, E1    +3.155, E3 +20594.179}
SPL {X  -160.000, Y  +652.103, Z    +0.000, E1   +11.247, E3 +20605.850}
SPL {X  -160.000, Y  +641.822, Z    +0.000, E1   +17.059, E3 +20625.223}
SPL {X  -160.000, Y  +631.293, Z    +0.000, E1   +20.354, E3 +20659.103}
SPL {X  -160.000, Y  +627.542, Z    +0.000, E1   +20.380, E3 +20680.510}
SPL {X  -160.000, Y  +623.532, Z    +0.000, E1   +20.378, E3 +20703.476}
SPL {X  -160.000, Y  +619.329, Z    +0.000, E1   +20.391, E3 +20727.513}
SPL {X  -160.000, Y  +614.967, Z    +0.000, E1   +20.392, E3 +20752.493}
SPL {X  -160.000, Y  +611.206, Z    +0.000, E1   +20.351, E3 +20774.165}
SPL {X  -160.000, Y  +607.824, Z    +0.000, E1   +20.354, E3 +20793.585}
SPL {X  -160.000, Y  +603.899, Z    +0.000, E1   +20.373, E3 +20816.035}
SPL {X  -160.000, Y  +599.617, Z    +0.000, E1   +20.384, E3 +20840.529}
SPL {X  -160.000, Y  +595.532, Z    +0.000, E1   +20.373, E3 +20863.890}
SPL {X  -160.000, Y  +591.705, Z    +0.000, E1   +20.373, E3 +20885.814}
SPL {X  -160.000, Y  +588.037, Z    +0.000, E1   +20.359, E3 +20906.901}
SPL {X  -160.000, Y  +584.320, Z    +0.000, E1   +20.364, E3 +20928.203}
SPL {X  -160.000, Y  +580.616, Z    +0.000, E1   +20.357, E3 +20949.430}
SPL {X  -160.000, Y  +577.083, Z    +0.000, E1   +20.358, E3 +20969.678}
SPL {X  -160.000, Y  +573.158, Z    +0.000, E1   +20.377, E3 +20992.131}
SPL {X  -160.000, Y  +568.802, Z    +0.000, E1   +20.385, E3 +21017.082}
SPL {X  -160.000, Y  +564.937, Z    +0.000, E1   +20.350, E3 +21039.303}
SPL {X  -160.000, Y  +561.213, Z    +0.000, E1   +20.372, E3 +21060.589}
SPL {X  -160.000, Y  +557.320, Z    +0.000, E1   +20.363, E3 +21082.916}
SPL {X  -160.000, Y  +553.712, Z    +0.000, E1   +20.355, E3 +21103.616}
SPL {X  -160.000, Y  +550.040, Z    +0.000, E1   +20.360, E3 +21124.654}
SPL {X  -160.000, Y  +546.180, Z    +0.000, E1   +20.370, E3 +21146.709}
SPL {X  -160.000, Y  +542.032, Z    +0.000, E1   +20.384, E3 +21170.448}
SPL {X  -160.000, Y  +537.870, Z    +0.000, E1   +20.372, E3 +21194.324}
SPL {X  -160.000, Y  +534.086, Z    +0.000, E1   +20.356, E3 +21216.078}
SPL {X  -160.000, Y  +530.164, Z    +0.000, E1   +20.382, E3 +21238.427}
SPL {X  -160.000, Y  +527.505, Z    +0.000, E1   +20.318, E3 +21253.801}
SPL {X  -160.000, Y  +511.620, Z    +0.000, E1   +28.365, E3 +21264.264}
SPL {X  -160.000, Y  +507.906, Z    +0.000, E1   +28.152, E3 +21280.659}
SPL {X  -160.000, Y  +506.085, Z    +0.000, E1   +26.146, E3 +21303.119}
SPL {X  -160.000, Y  +504.342, Z    +0.000, E1   +24.109, E3 +21326.634}
SPL {X  -160.000, Y  +503.002, Z    +0.000, E1   +22.325, E3 +21347.639}
SPL {X  -160.000, Y  +500.783, Z    +0.000, E1   +21.421, E3 +21367.229}
SPL {X  -160.000, Y  +497.229, Z    +0.000, E1   +21.403, E3 +21386.537}
SPL {X  -160.000, Y  +493.901, Z    +0.000, E1   +21.409, E3 +21404.556}
SPL {X  -160.000, Y  +490.791, Z    +0.000, E1   +21.400, E3 +21421.429}
SPL {X  -160.000, Y  +487.647, Z    +0.000, E1   +21.401, E3 +21438.475}
SPL {X  -160.000, Y  +484.273, Z    +0.000, E1   +21.408, E3 +21456.755}
SPL {X  -160.000, Y  +481.093, Z    +0.000, E1   +21.389, E3 +21474.064}
SPL {X  -160.000, Y  +478.021, Z    +0.000, E1   +21.401, E3 +21490.671}
SPL {X  -160.000, Y  +474.639, Z    +0.000, E1   +21.410, E3 +21508.962}
SPL {X  -160.000, Y  +471.343, Z    +0.000, E1   +21.399, E3 +21526.864}
SPL {X  -160.000, Y  +468.133, Z    +0.000, E1   +21.402, E3 +21544.255}
SPL {X  -160.000, Y  +464.638, Z    +0.000, E1   +21.421, E3 +21563.105}
SPL {X  -160.000, Y  +461.045, Z    +0.000, E1   +21.424, E3 +21582.518}
SPL {X  -160.000, Y  +457.606, Z    +0.000, E1   +21.413, E3 +21601.228}
SPL {X  -160.000, Y  +454.417, Z    +0.000, E1   +21.401, E3 +21618.537}
SPL {X  -160.000, Y  +451.425, Z    +0.000, E1   +21.404, E3 +21634.759}
SPL {X  -160.000, Y  +448.039, Z    +0.000, E1   +21.417, E3 +21653.051}
SPL {X  -160.000, Y  +444.787, Z    +0.000, E1   +21.414, E3 +21670.607}
SPL {X  -160.000, Y  +441.637, Z    +0.000, E1   +21.431, E3 +21687.585}
SPL {X  -160.000, Y  +438.199, Z    +0.000, E1   +21.432, E3 +21706.189}
SPL {X  -160.000, Y  +434.875, Z    +0.000, E1   +21.424, E3 +21724.228}
SPL {X  -160.000, Y  +431.689, Z    +0.000, E1   +21.423, E3 +21741.477}
SPL {X  -160.000, Y  +428.451, Z    +0.000, E1   +21.430, E3 +21758.956}
SPL {X  -160.000, Y  +425.120, Z    +0.000, E1   +21.430, E3 +21777.021}
SPL {X  -160.000, Y  +421.671, Z    +0.000, E1   +21.430, E3 +21795.705}
SPL {X  -160.000, Y  +418.225, Z    +0.000, E1   +21.425, E3 +21814.386}
SPL {X  -160.000, Y  +414.956, Z    +0.000, E1   +21.424, E3 +21832.067}
SPL {X  -160.000, Y  +411.834, Z    +0.000, E1   +21.420, E3 +21848.985}
SPL {X  -160.000, Y  +408.570, Z    +0.000, E1   +21.432, E3 +21866.594}
SPL {X  -160.000, Y  +405.237, Z    +0.000, E1   +21.432, E3 +21884.623}
SPL {X  -160.000, Y  +402.004, Z    +0.000, E1   +21.424, E3 +21902.198}
SPL {X  -160.000, Y  +398.626, Z    +0.000, E1   +21.425, E3 +21920.504}
SPL {X  -160.000, Y  +395.405, Z    +0.000, E1   +21.422, E3 +21937.922}
SPL {X  -160.000, Y  +392.641, Z    +0.000, E1   +21.407, E3 +21952.920}
SPL {X  -159.989, Y  +390.129, Z    +0.000, E1   +21.406, E3 +21966.561}
SPL {X  -159.932, Y  +387.337, Z    +0.000, E1   +21.403, E3 +21981.757}
SPL {X  -159.823, Y  +384.478, Z    +0.000, E1   +21.379, E3 +21997.420}
SPL {X  -159.660, Y  +381.581, Z    +0.000, E1   +21.363, E3 +22013.308}
SPL {X  -159.452, Y  +378.773, Z    +0.000, E1   +21.330, E3 +22028.755}
SPL {X  -159.222, Y  +376.244, Z    +0.000, E1   +21.297, E3 +22042.717}
SPL {X  -158.814, Y  +372.556, Z    +0.000, E1   +21.316, E3 +22062.984}
SPL {X  -158.301, Y  +368.743, Z    +0.000, E1   +21.199, E3 +22084.306}
SPL {X  -157.981, Y  +366.660, Z    +0.000, E1   +19.986, E3 +22107.273}
ENDSPLINE

SPLINE
SPL {X  -158.491, Y  +370.077, Z    +0.000, E1   +15.910, E3 +22132.286}
SPL {X  -159.771, Y  +383.450, Z    +0.000, E1    +6.314, E3 +22155.442}
SPL {X  -160.000, Y  +392.463, Z    +0.000, E1    +0.112, E3 +22161.949}
SPL {X  -160.000, Y  +399.874, Z    +0.000, E1    -5.508, E3 +22166.451}
SPL {X  -160.000, Y  +411.622, Z    +0.000, E1   -13.815, E3 +22178.571}
SPL {X  -160.000, Y  +419.836, Z    +0.000, E1   -18.198, E3 +22193.745}
SPL {X  -160.000, Y  +430.523, Z    +0.000, E1   -21.710, E3 +22223.945}
SPL {X  -160.000, Y  +433.426, Z    +0.000, E1   -21.735, E3 +22239.359}
SPL {X  -160.000, Y  +436.131, Z    +0.000, E1   -21.710, E3 +22253.834}
SPL {X  -160.000, Y  +439.046, Z    +0.000, E1   -21.732, E3 +22269.327}
SPL {X  -160.000, Y  +442.009, Z    +0.000, E1   -21.719, E3 +22285.149}
SPL {X  -160.000, Y  +444.891, Z    +0.000, E1   -21.724, E3 +22300.505}
SPL {X  -160.000, Y  +449.017, Z    +0.000, E1   -21.792, E3 +22322.297}
SPL {X  -160.000, Y  +452.864, Z    +0.000, E1   -21.730, E3 +22342.915}
SPL {X  -160.000, Y  +455.470, Z    +0.000, E1   -21.722, E3 +22356.803}
SPL {X  -160.000, Y  +458.295, Z    +0.000, E1   -21.738, E3 +22371.824}
SPL {X  -160.000, Y  +461.133, Z    +0.000, E1   -21.720, E3 +22387.007}
SPL {X  -160.000, Y  +464.458, Z    +0.000, E1   -21.770, E3 +22404.526}
SPL {X  -160.000, Y  +468.250, Z    +0.000, E1   -21.764, E3 +22424.679}
SPL {X  -160.000, Y  +472.226, Z    +0.000, E1   -21.782, E3 +22445.837}
SPL {X  -160.000, Y  +476.333, Z    +0.000, E1   -21.767, E3 +22467.752}
SPL {X  -160.000, Y  +480.244, Z    +0.000, E1   -21.765, E3 +22488.616}
SPL {X  -160.000, Y  +484.301, Z    +0.000, E1   -21.775, E3 +22510.145}
SPL {X  -160.000, Y  +488.201, Z    +0.000, E1   -21.768, E3 +22530.905}
SPL {X  -160.000, Y  +492.394, Z    +0.000, E1   -21.802, E3 +22553.079}
SPL {X  -160.000, Y  +496.781, Z    +0.000, E1   -21.798, E3 +22576.390}
SPL {X  -160.000, Y  +501.083, Z    +0.000, E1   -21.796, E3 +22599.320}
SPL {X  -160.000, Y  +504.917, Z    +0.000, E1   -21.764, E3 +22619.825}
SPL {X  -160.000, Y  +508.886, Z    +0.000, E1   -21.791, E3 +22640.911}
SPL {X  -160.000, Y  +513.057, Z    +0.000, E1   -21.767, E3 +22663.219}
SPL {X  -160.000, Y  +517.221, Z    +0.000, E1   -21.778, E3 +22685.371}
SPL {X  -160.000, Y  +521.677, Z    +0.000, E1   -21.781, E3 +22709.132}
SPL {X  -160.000, Y  +525.729, Z    +0.000, E1   -21.753, E3 +22730.772}
SPL {X  -160.000, Y  +529.456, Z    +0.000, E1   -21.766, E3 +22750.551}
SPL {X  -160.000, Y  +533.608, Z    +0.000, E1   -21.776, E3 +22772.681}
SPL {X  -160.000, Y  +538.227, Z    +0.000, E1   -21.794, E3 +22797.214}
SPL {X  -160.000, Y  +542.483, Z    +0.000, E1   -21.764, E3 +22819.939}
SPL {X  -160.000, Y  +546.194, Z    +0.000, E1   -21.754, E3 +22839.756}
SPL {X  -160.000, Y  +550.131, Z    +0.000, E1   -21.771, E3 +22860.691}
SPL {X  -160.000, Y  +554.462, Z    +0.000, E1   -21.777, E3 +22883.745}
SPL {X  -160.000, Y  +558.542, Z    +0.000, E1   -21.758, E3 +22905.518}
SPL {X  -160.000, Y  +562.615, Z    +0.000, E1   -21.776, E3 +22927.174}
SPL {X  -160.000, Y  +566.764, Z    +0.000, E1   -21.764, E3 +22949.299}
SPL {X  -160.000, Y  +570.657, Z    +0.000, E1   -21.758, E3 +22970.046}
SPL {X  -160.000, Y  +574.688, Z    +0.000, E1   -21.771, E3 +22991.489}
SPL {X  -160.000, Y  +578.864, Z    +0.000, E1   -21.770, E3 +23013.740}
SPL {X  -160.000, Y  +582.807, Z    +0.000, E1   -21.754, E3 +23034.794}
SPL {X  -160.000, Y  +586.993, Z    +0.000, E1   -21.779, E3 +23057.030}
SPL {X  -160.000, Y  +591.368, Z    +0.000, E1   -21.775, E3 +23080.317}
SPL {X  -160.000, Y  +595.703, Z    +0.000, E1   -21.775, E3 +23103.426}
SPL {X  -160.000, Y  +599.558, Z    +0.000, E1   -21.748, E3 +23124.003}
SPL {X  -160.000, Y  +603.126, Z    +0.000, E1   -21.757, E3 +23142.983}
SPL {X  -160.000, Y  +607.107, Z    +0.000, E1   -21.766, E3 +23164.208}
SPL {X  -160.000, Y  +611.246, Z    +0.000, E1   -21.760, E3 +23186.281}
SPL {X  -160.000, Y  +615.151, Z    +0.000, E1   -21.752, E3 +23207.095}
SPL {X  -160.000, Y  +618.728, Z    +0.000, E1   -21.747, E3 +23226.157}
SPL {X  -160.000, Y  +622.318, Z    +0.000, E1   -21.753, E3 +23245.272}
SPL {X  -160.000, Y  +625.877, Z    +0.000, E1   -21.745, E3 +23264.250}
SPL {X  -160.000, Y  +629.892, Z    +0.000, E1   -21.777, E3 +23285.574}
SPL {X  -160.000, Y  +634.024, Z    +0.000, E1   -21.756, E3 +23307.624}
SPL {X  -160.000, Y  +637.661, Z    +0.000, E1   -21.748, E3 +23327.015}
SPL {X  -160.000, Y  +641.244, Z    +0.000, E1   -21.752, E3 +23346.085}
SPL {X  -160.000, Y  +645.120, Z    +0.000, E1   -21.762, E3 +23366.718}
SPL {X  -160.000, Y  +649.214, Z    +0.000, E1   -21.766, E3 +23388.506}
SPL {X  -160.000, Y  +653.188, Z    +0.000, E1   -21.771, E3 +23409.569}
SPL {X  -160.000, Y  +656.905, Z    +0.000, E1   -21.769, E3 +23429.344}
SPL {X  -160.000, Y  +660.685, Z    +0.000, E1   -21.769, E3 +23449.512}
SPL {X  -160.000, Y  +664.985, Z    +0.000, E1   -21.790, E3 +23472.365}
SPL {X  -159.993, Y  +669.170, Z    +0.000, E1   -21.763, E3 +23494.723}
SPL {X  -159.916, Y  +672.869, Z    +0.000, E1   -21.755, E3 +23514.468}
SPL {X  -159.752, Y  +676.610, Z    +0.000, E1   -21.740, E3 +23534.543}
SPL {X  -159.478, Y  +680.618, Z    +0.000, E1   -21.719, E3 +23556.142}
SPL {X  -159.108, Y  +684.576, Z    +0.000, E1   -21.664, E3 +23577.611}
SPL {X  -158.638, Y  +688.530, Z    +0.000, E1   -21.617, E3 +23599.133}
SPL {X  -158.097, Y  +692.303, Z    +0.000, E1   -21.529, E3 +23619.851}
ENDSPLINE

SPLINE
SPL {X  -158.264, Y  +691.203, Z    +0.000, E1   -17.264, E3 +23656.596}
SPL {X  -159.000, Y  +685.560, Z    +0.000, E1   -12.398, E3 +23677.771}
SPL {X  -159.924, Y  +672.625, Z    +0.000, E1    -3.689, E3 +23692.788}
SPL {X  -160.000, Y  +663.203, Z    +0.000, E1    +3.155, E3 +23699.443}
SPL {X  -160.000, Y  +652.103, Z    +0.000, E1   +11.247, E3 +23711.113}
SPL {X  -160.000, Y  +641.822, Z    +0.000, E1   +17.059, E3 +23730.487}
SPL {X  -160.000, Y  +631.293, Z    +0.000, E1   +20.354, E3 +23764.366}
SPL {X  -160.000, Y  +627.542, Z    +0.000, E1   +20.380, E3 +23785.773}
SPL {X  -160.000, Y  +623.532, Z    +0.000, E1   +20.378, E3 +23808.739}
SPL {X  -160.000, Y  +619.329, Z    +0.000, E1   +20.391, E3 +23832.777}
SPL {X  -160.000, Y  +614.967, Z    +0.000, E1   +20.392, E3 +23857.756}
SPL {X  -160.000, Y  +611.206, Z    +0.000, E1   +20.351, E3 +23879.428}
SPL {X  -160.000, Y  +607.824, Z    +0.000, E1   +20.354, E3 +23898.849}
SPL {X  -160.000, Y  +603.899, Z    +0.000, E1   +20.373, E3 +23921.299}
SPL {X  -160.000, Y  +599.617, Z    +0.000, E1   +20.384, E3 +23945.793}
SPL {X  -160.000, Y  +595.532, Z    +0.000, E1   +20.373, E3 +23969.153}
SPL {X  -160.000, Y  +591.705, Z    +0.000, E1   +20.373, E3 +23991.078}
SPL {X  -160.000, Y  +588.037, Z    +0.000, E1   +20.359, E3 +24012.165}
SPL {X  -160.000, Y  +584.320, Z    +0.000, E1   +20.364, E3 +24033.467}
SPL {X  -160.000, Y  +580.616, Z    +0.000, E1   +20.357, E3 +24054.693}
SPL {X  -160.000, Y  +577.083, Z    +0.000, E1   +20.358, E3 +24074.942}
SPL {X  -160.000, Y  +573.158, Z    +0.000, E1   +20.377, E3 +24097.394}
SPL {X  -160.000, Y  +568.802, Z    +0.000, E1   +20.385, E3 +24122.346}
SPL {X  -160.000, Y  +564.937, Z    +0.000, E1   +20.350, E3 +24144.566}
SPL {X  -160.000, Y  +561.213, Z    +0.000, E1   +20.372, E3 +24165.853}
SPL {X  -160.000, Y  +557.320, Z    +0.000, E1   +20.363, E3 +24188.180}
SPL {X  -160.000, Y  +553.712, Z    +0.000, E1   +20.355, E3 +24208.879}
SPL {X  -160.000, Y  +550.040, Z    +0.000, E1   +20.360, E3 +24229.917}
SPL {X  -160.000, Y  +546.180, Z    +0.000, E1   +20.370, E3 +24251.973}
SPL {X  -160.000, Y  +542.032, Z    +0.000, E1   +20.384, E3 +24275.712}
SPL {X  -160.000, Y  +537.870, Z    +0.000, E1   +20.372, E3 +24299.587}
SPL {X  -160.000, Y  +534.086, Z    +0.000, E1   +20.356, E3 +24321.341}
SPL {X  -160.000, Y  +530.164, Z    +0.000, E1   +20.382, E3 +24343.691}
SPL {X  -160.000, Y  +527.505, Z    +0.000, E1   +20.318, E3 +24359.065}
SPL {X  -160.000, Y  +511.620, Z    +0.000, E1   +28.365, E3 +24369.528}
SPL {X  -160.000, Y  +507.906, Z    +0.000, E1   +28.152, E3 +24385.923}
SPL {X  -160.000, Y  +506.085, Z    +0.000, E1   +26.146, E3 +24408.382}
SPL {X  -160.000, Y  +504.342, Z    +0.000, E1   +24.109, E3 +24431.897}
SPL {X  -160.000, Y  +503.002, Z    +0.000, E1   +22.325, E3 +24452.903}
SPL {X  -160.000, Y  +500.783, Z    +0.000, E1   +21.421, E3 +24472.492}
SPL {X  -160.000, Y  +497.229, Z    +0.000, E1   +21.403, E3 +24491.800}
SPL {X  -160.000, Y  +493.901, Z    +0.000, E1   +21.409, E3 +24509.819}
SPL {X  -160.000, Y  +490.791, Z    +0.000, E1   +21.400, E3 +24526.692}
SPL {X  -160.000, Y  +487.647, Z    +0.000, E1   +21.401, E3 +24543.738}
SPL {X  -160.000, Y  +484.273, Z    +0.000, E1   +21.408, E3 +24562.018}
SPL {X  -160.000, Y  +481.093, Z    +0.000, E1   +21.389, E3 +24579.327}
SPL {X  -160.000, Y  +478.021, Z    +0.000, E1   +21.401, E3 +24595.934}
SPL {X  -160.000, Y  +474.639, Z    +0.000, E1   +21.410, E3 +24614.225}
SPL {X  -160.000, Y  +471.343, Z    +0.000, E1   +21.399, E3 +24632.127}
SPL {X  -160.000, Y  +468.133, Z    +0.000, E1   +21.402, E3 +24649.519}
SPL {X  -160.000, Y  +464.638, Z    +0.000, E1   +21.421, E3 +24668.368}
SPL {X  -160.000, Y  +461.045, Z    +0.000, E1   +21.424, E3 +24687.782}
SPL {X  -160.000, Y  +457.606, Z    +0.000, E1   +21.413, E3 +24706.492}
SPL {X  -160.000, Y  +454.417, Z    +0.000, E1   +21.401, E3 +24723.800}
SPL {X  -160.000, Y  +451.425, Z    +0.000, E1   +21.404, E3 +24740.022}
SPL {X  -160.000, Y  +448.039, Z    +0.000, E1   +21.417, E3 +24758.315}
SPL {X  -160.000, Y  +444.787, Z    +0.000, E1   +21.414, E3 +24775.870}
SPL {X  -160.000, Y  +441.637, Z    +0.000, E1   +21.431, E3 +24792.848}
SPL {X  -160.000, Y  +438.199, Z    +0.000, E1   +21.432, E3 +24811.452}
SPL {X  -160.000, Y  +434.875, Z    +0.000, E1   +21.424, E3 +24829.492}
SPL {X  -160.000, Y  +431.689, Z    +0.000, E1   +21.423, E3 +24846.740}
SPL {X  -160.000, Y  +428.451, Z    +0.000, E1   +21.430, E3 +24864.220}
SPL {X  -160.000, Y  +425.120, Z    +0.000, E1   +21.430, E3 +24882.284}
SPL {X  -160.000, Y  +421.671, Z    +0.000, E1   +21.430, E3 +24900.968}
SPL {X  -160.000, Y  +418.225, Z    +0.000, E1   +21.425, E3 +24919.650}
SPL {X  -160.000, Y  +414.956, Z    +0.000, E1   +21.424, E3 +24937.330}
SPL {X  -160.000, Y  +411.834, Z    +0.000, E1   +21.420, E3 +24954.249}
SPL {X  -160.000, Y  +408.570, Z    +0.000, E1   +21.432, E3 +24971.858}
SPL {X  -160.000, Y  +405.237, Z    +0.000, E1   +21.432, E3 +24989.886}
SPL {X  -160.000, Y  +402.004, Z    +0.000, E1   +21.424, E3 +25007.462}
SPL {X  -160.000, Y  +398.626, Z    +0.000, E1   +21.425, E3 +25025.768}
SPL {X  -160.000, Y  +395.405, Z    +0.000, E1   +21.422, E3 +25043.185}
SPL {X  -160.000, Y  +392.641, Z    +0.000, E1   +21.407, E3 +25058.183}
SPL {X  -159.989, Y  +390.129, Z    +0.000, E1   +21.406, E3 +25071.824}
SPL {X  -159.932, Y  +387.337, Z    +0.000, E1   +21.403, E3 +25087.020}
SPL {X  -159.823, Y  +384.478, Z    +0.000, E1   +21.379, E3 +25102.683}
SPL {X  -159.660, Y  +381.581, Z    +0.000, E1   +21.363, E3 +25118.571}
SPL {X  -159.452, Y  +378.773, Z    +0.000, E1   +21.330, E3 +25134.018}
SPL {X  -159.222, Y  +376.244, Z    +0.000, E1   +21.297, E3 +25147.980}
SPL {X  -158.814, Y  +372.556, Z    +0.000, E1   +21.316, E3 +25168.247}
SPL {X  -158.301, Y  +368.743, Z    +0.000, E1   +21.199, E3 +25189.569}
SPL {X  -157.981, Y  +366.660, Z    +0.000, E1   +19.986, E3 +25212.537}
ENDSPLINE

